// Mitsubishi GX Works2 project: GCP-75A2RB-(SECS)20220112   PLC: Q03UDV

PROGRAM 01INITI
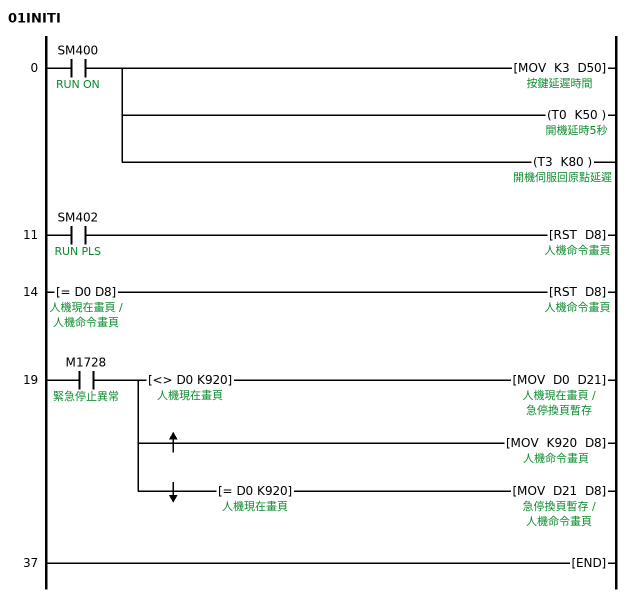
0     LD      SM400  ; RUN ON
      MOV     K3 D50  ; 按鍵延遲時間
      OUT     T0 K50  ; 開機延時5秒
      OUT     T3 K80  ; 開機伺服回原點延遲
11    LD      SM402  ; RUN PLS
      RST     D8  ; 人機命令畫頁
14    LD=     D0 D8  ; 人機現在畫頁 / 人機命令畫頁
      RST     D8  ; 人機命令畫頁
19    LD      M1728  ; 緊急停止異常
      MPS
      AND<>   D0 K920  ; 人機現在畫頁
      MOV     D0 D21  ; 急停換頁暫存
      MRD
      MEP
      MOV     K920 D8
      MPP
      MEF
      AND=    D0 K920  ; 人機現在畫頁
      MOV     D21 D8
37    END
END_PROGRAM

PROGRAM 02FUNC
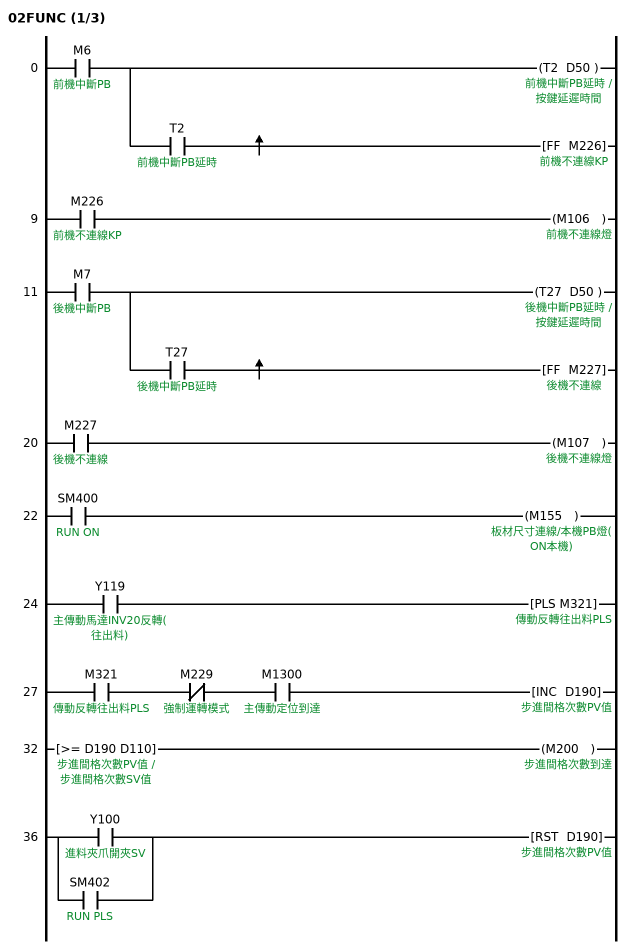
0     LD      M6  ; 前機中斷PB
      OUT     T2 D50  ; 前機中斷PB延時 / 按鍵延遲時間
      AND     T2  ; 前機中斷PB延時
      MEP
      FF      M226  ; 前機不連線KP
9     LD      M226  ; 前機不連線KP
      OUT     M106  ; 前機不連線燈
11    LD      M7  ; 後機中斷PB
      OUT     T27 D50  ; 後機中斷PB延時 / 按鍵延遲時間
      AND     T27  ; 後機中斷PB延時
      MEP
      FF      M227  ; 後機不連線
20    LD      M227  ; 後機不連線
      OUT     M107  ; 後機不連線燈
22    LD      SM400  ; RUN ON
      OUT     M155  ; 板材尺寸連線/本機PB燈(ON本機)
24    LD      Y119  ; 主傳動馬達INV20反轉(往出料)
      PLS     M321  ; 傳動反轉往出料PLS
27    LD      M321  ; 傳動反轉往出料PLS
      ANI     M229  ; 強制運轉模式
      AND     M1300  ; 主傳動定位到達
      INC     D190  ; 步進間格次數PV值
32    LD>=    D190 D110  ; 步進間格次數PV值 / 步進間格次數SV值
      OUT     M200  ; 步進間格次數到達
36    LD      Y100  ; 進料夾爪開夾SV
      OR      SM402  ; RUN PLS
      RST     D190  ; 步進間格次數PV值
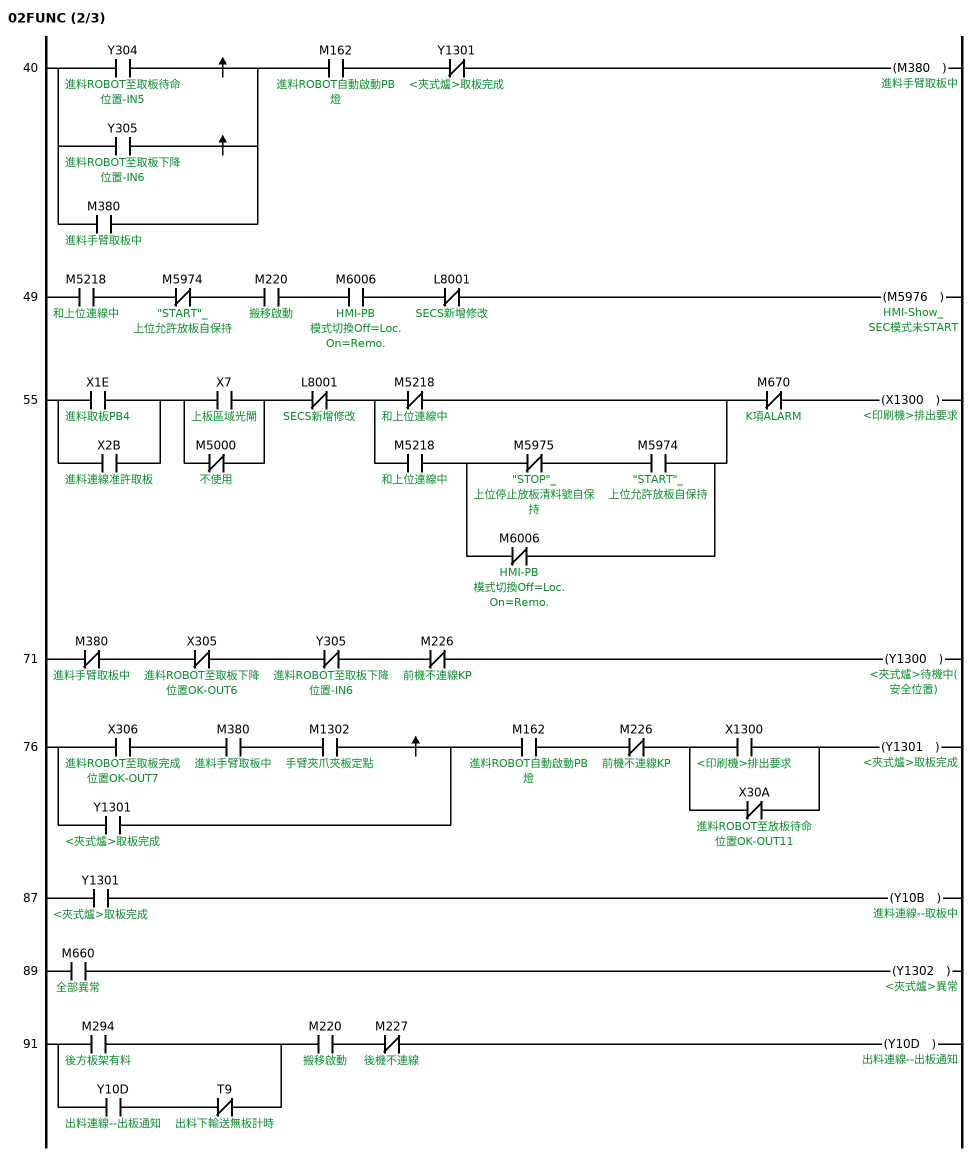
40    LD      Y304  ; 進料ROBOT至取板待命位置-IN5
      MEP
      LD      Y305  ; 進料ROBOT至取板下降位置-IN6
      MEP
      ORB
      OR      M380  ; 進料手臂取板中
      AND     M162  ; 進料ROBOT自動啟動PB燈
      ANI     Y1301  ; <夾式爐>取板完成
      OUT     M380  ; 進料手臂取板中
49    LD      M5218  ; 和上位連線中
      ANI     M5974  ; "START"_上位允許放板自保持
      AND     M220  ; 搬移啟動
      AND     M6006  ; HMI-PB  模式切換Off=Loc.On=Remo.
      ANI     L8001  ; SECS新增修改
      OUT     M5976  ; HMI-Show_SEC模式未START
55    LD      X1E  ; 進料取板PB4
      OR      X2B  ; 進料連線准許取板
      LD      X7  ; 上板區域光閘
      ORI     M5000  ; 不使用
      ANB
      ANI     L8001  ; SECS新增修改
      LDI     M5218  ; 和上位連線中
      LD      M5218  ; 和上位連線中
      LDI     M5975  ; "STOP"_ 上位停止放板清料號自保持
      AND     M5974  ; "START"_上位允許放板自保持
      ORI     M6006  ; HMI-PB  模式切換Off=Loc.On=Remo.
      ANB
      ORB
      ANB
      ANI     M670  ; K項ALARM
      OUT     X1300  ; <印刷機>排出要求
71    LDI     M380  ; 進料手臂取板中
      ANI     X305  ; 進料ROBOT至取板下降位置OK-OUT6
      ANI     Y305  ; 進料ROBOT至取板下降位置-IN6
      ANI     M226  ; 前機不連線KP
      OUT     Y1300  ; <夾式爐>待機中(安全位置)
76    LD      X306  ; 進料ROBOT至取板完成位置OK-OUT7
      AND     M380  ; 進料手臂取板中
      AND     M1302  ; 手臂夾爪夾板定點
      MEP
      OR      Y1301  ; <夾式爐>取板完成
      AND     M162  ; 進料ROBOT自動啟動PB燈
      ANI     M226  ; 前機不連線KP
      LD      X1300  ; <印刷機>排出要求
      ORI     X30A  ; 進料ROBOT至放板待命位置OK-OUT11
      ANB
      OUT     Y1301  ; <夾式爐>取板完成
87    LD      Y1301  ; <夾式爐>取板完成
      OUT     Y10B  ; 進料連線--取板中
89    LD      M660  ; 全部異常
      OUT     Y1302  ; <夾式爐>異常
91    LD      M294  ; 後方板架有料
      LD      Y10D  ; 出料連線--出板通知
      ANI     T9  ; 出料下輸送無板計時
      ORB
      AND     M220  ; 搬移啟動
      ANI     M227  ; 後機不連線
      OUT     Y10D  ; 出料連線--出板通知
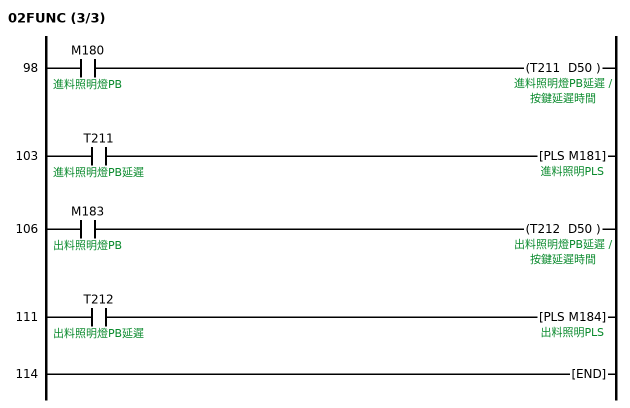
98    LD      M180  ; 進料照明燈PB
      OUT     T211 D50  ; 進料照明燈PB延遲 / 按鍵延遲時間
103   LD      T211  ; 進料照明燈PB延遲
      PLS     M181  ; 進料照明PLS
106   LD      M183  ; 出料照明燈PB
      OUT     T212 D50  ; 出料照明燈PB延遲 / 按鍵延遲時間
111   LD      T212  ; 出料照明燈PB延遲
      PLS     M184  ; 出料照明PLS
114   END
END_PROGRAM

PROGRAM 03ORIGIN
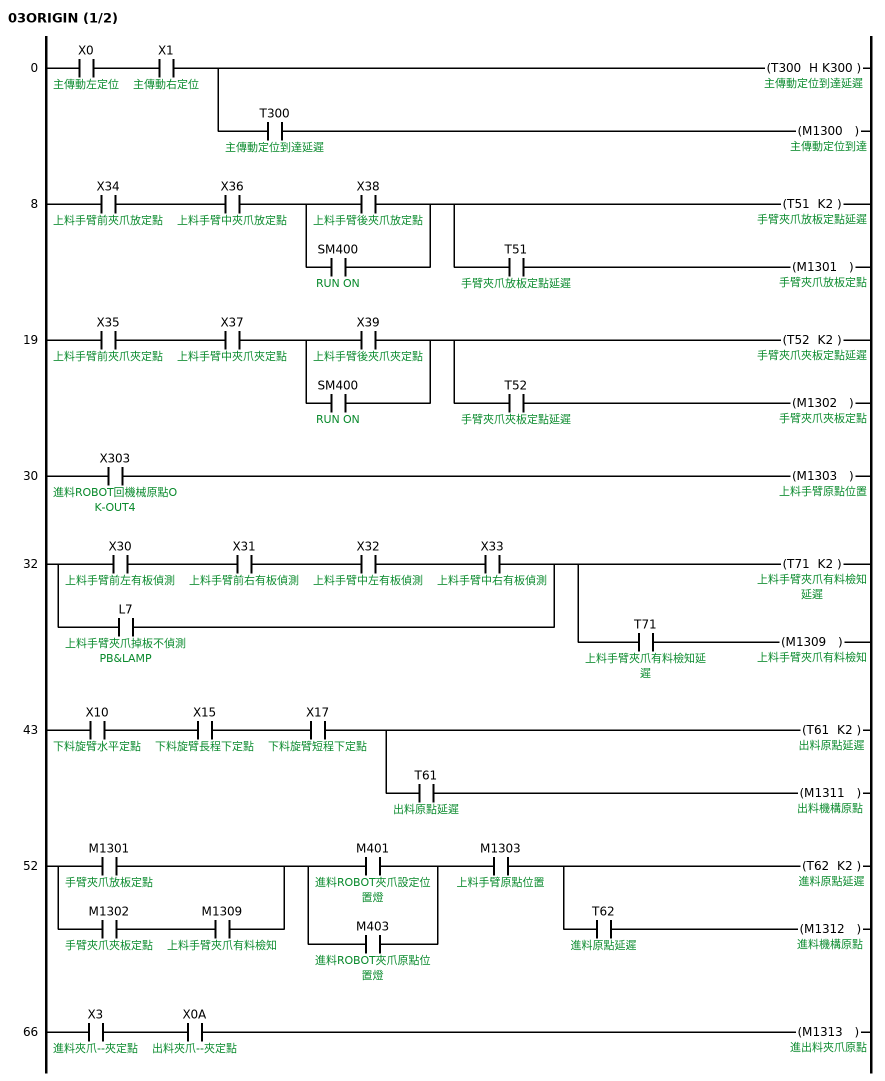
0     LD      X0  ; 主傳動左定位
      AND     X1  ; 主傳動右定位
      OUTH    T300 K300  ; 主傳動定位到達延遲
      AND     T300  ; 主傳動定位到達延遲
      OUT     M1300  ; 主傳動定位到達
8     LD      X34  ; 上料手臂前夾爪放定點
      AND     X36  ; 上料手臂中夾爪放定點
      LD      X38  ; 上料手臂後夾爪放定點
      OR      SM400  ; RUN ON
      ANB
      OUT     T51 K2  ; 手臂夾爪放板定點延遲
      AND     T51  ; 手臂夾爪放板定點延遲
      OUT     M1301  ; 手臂夾爪放板定點
19    LD      X35  ; 上料手臂前夾爪夾定點
      AND     X37  ; 上料手臂中夾爪夾定點
      LD      X39  ; 上料手臂後夾爪夾定點
      OR      SM400  ; RUN ON
      ANB
      OUT     T52 K2  ; 手臂夾爪夾板定點延遲
      AND     T52  ; 手臂夾爪夾板定點延遲
      OUT     M1302  ; 手臂夾爪夾板定點
30    LD      X303  ; 進料ROBOT回機械原點OK-OUT4
      OUT     M1303  ; 上料手臂原點位置
32    LD      X30  ; 上料手臂前左有板偵測
      AND     X31  ; 上料手臂前右有板偵測
      AND     X32  ; 上料手臂中左有板偵測
      AND     X33  ; 上料手臂中右有板偵測
      OR      L7  ; 上料手臂夾爪掉板不偵測PB&LAMP
      OUT     T71 K2  ; 上料手臂夾爪有料檢知延遲
      AND     T71  ; 上料手臂夾爪有料檢知延遲
      OUT     M1309  ; 上料手臂夾爪有料檢知
43    LD      X10  ; 下料旋臂水平定點
      AND     X15  ; 下料旋臂長程下定點
      AND     X17  ; 下料旋臂短程下定點
      OUT     T61 K2  ; 出料原點延遲
      AND     T61  ; 出料原點延遲
      OUT     M1311  ; 出料機構原點
52    LD      M1301  ; 手臂夾爪放板定點
      LD      M1302  ; 手臂夾爪夾板定點
      AND     M1309  ; 上料手臂夾爪有料檢知
      ORB
      LD      M401  ; 進料ROBOT夾爪設定位置燈
      OR      M403  ; 進料ROBOT夾爪原點位置燈
      ANB
      AND     M1303  ; 上料手臂原點位置
      OUT     T62 K2  ; 進料原點延遲
      AND     T62  ; 進料原點延遲
      OUT     M1312  ; 進料機構原點
66    LD      X3  ; 進料夾爪--夾定點
      AND     X0A  ; 出料夾爪--夾定點
      OUT     M1313  ; 進出料夾爪原點
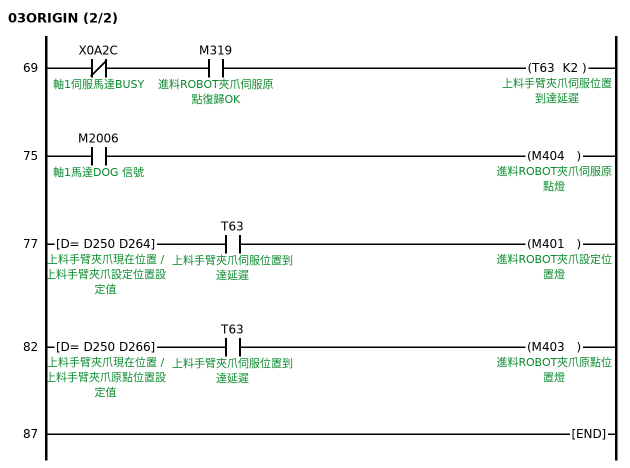
69    LDI     X0A2C  ; 軸1伺服馬達BUSY
      AND     M319  ; 進料ROBOT夾爪伺服原點復歸OK
      OUT     T63 K2  ; 上料手臂夾爪伺服位置到達延遲
75    LD      M2006  ; 軸1馬達DOG 信號
      OUT     M404  ; 進料ROBOT夾爪伺服原點燈
77    LDD=    D250 D264  ; 上料手臂夾爪現在位置 / 上料手臂夾爪設定位置設定值
      AND     T63  ; 上料手臂夾爪伺服位置到達延遲
      OUT     M401  ; 進料ROBOT夾爪設定位置燈
82    LDD=    D250 D266  ; 上料手臂夾爪現在位置 / 上料手臂夾爪原點位置設定值
      AND     T63  ; 上料手臂夾爪伺服位置到達延遲
      OUT     M403  ; 進料ROBOT夾爪原點位置燈
87    END
END_PROGRAM

PROGRAM 04LOAD
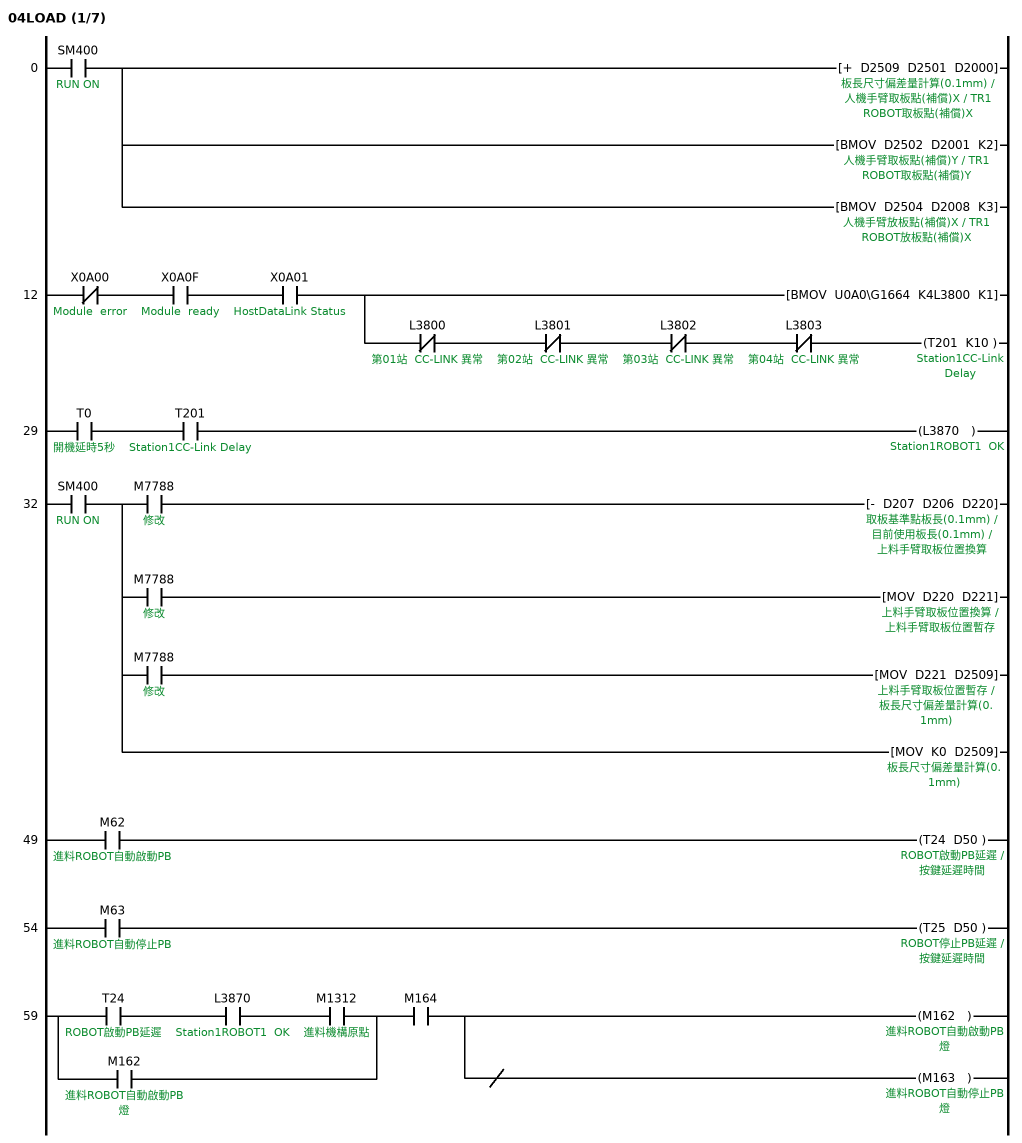
0     LD      SM400  ; RUN ON
      +       D2509 D2501 D2000  ; 板長尺寸偏差量計算(0.1mm) / 人機手臂取板點(補償)X / TR1 ROBOT取板點(補償)X
      BMOV    D2502 D2001 K2  ; 人機手臂取板點(補償)Y / TR1 ROBOT取板點(補償)Y
      BMOV    D2504 D2008 K3  ; 人機手臂放板點(補償)X / TR1 ROBOT放板點(補償)X
12    LDI     X0A00  ; Module  error
      AND     X0A0F  ; Module  ready
      AND     X0A01  ; HostDataLink Status
      BMOV    U0A0\G1664 K4L3800 K1  ; 第01站  CC-LINK 異常
      ANI     L3800  ; 第01站  CC-LINK 異常
      ANI     L3801  ; 第02站  CC-LINK 異常
      ANI     L3802  ; 第03站  CC-LINK 異常
      ANI     L3803  ; 第04站  CC-LINK 異常
      OUT     T201 K10  ; Station1CC-Link Delay
29    LD      T0  ; 開機延時5秒
      AND     T201  ; Station1CC-Link Delay
      OUT     L3870  ; Station1ROBOT1  OK
32    LD      SM400  ; RUN ON
      MPS
      AND     M7788  ; 修改
      -       D207 D206 D220  ; 取板基準點板長(0.1mm) / 目前使用板長(0.1mm) / 上料手臂取板位置換算
      MRD
      AND     M7788  ; 修改
      MOV     D220 D221  ; 上料手臂取板位置暫存
      MRD
      AND     M7788  ; 修改
      MOV     D221 D2509
      MPP
      MOV     K0 D2509
49    LD      M62  ; 進料ROBOT自動啟動PB
      OUT     T24 D50  ; ROBOT啟動PB延遲 / 按鍵延遲時間
54    LD      M63  ; 進料ROBOT自動停止PB
      OUT     T25 D50  ; ROBOT停止PB延遲 / 按鍵延遲時間
59    LD      T24  ; ROBOT啟動PB延遲
      AND     L3870  ; Station1ROBOT1  OK
      AND     M1312  ; 進料機構原點
      OR      M162  ; 進料ROBOT自動啟動PB燈
      AND     M164
      OUT     M162  ; 進料ROBOT自動啟動PB燈
      INV
      OUT     M163  ; 進料ROBOT自動停止PB燈
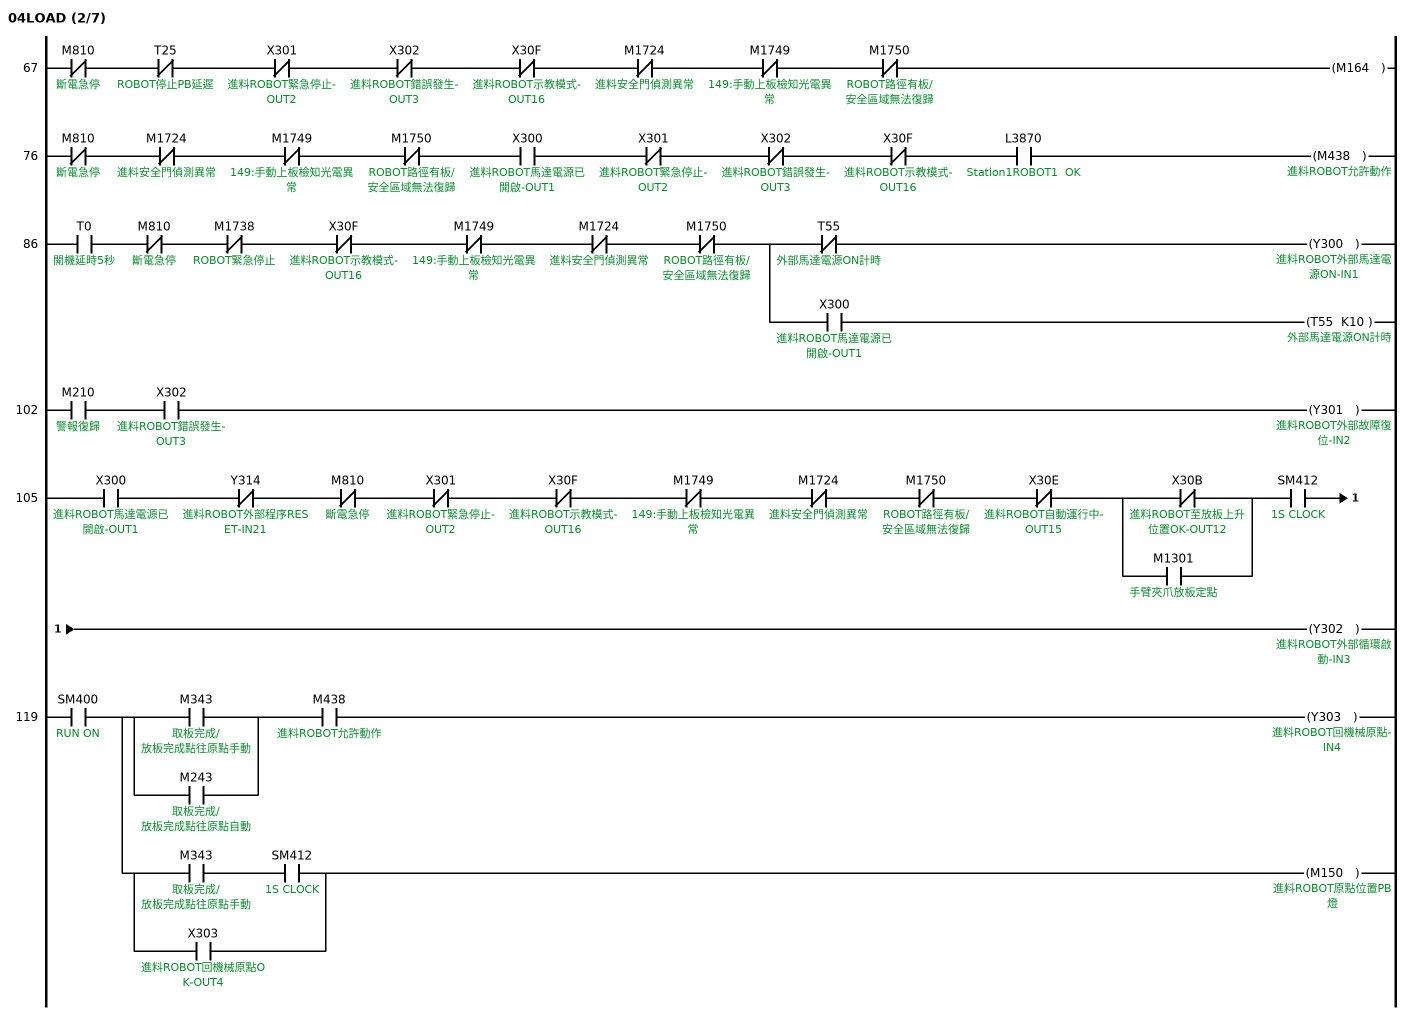
67    LDI     M810  ; 斷電急停
      ANI     T25  ; ROBOT停止PB延遲
      ANI     X301  ; 進料ROBOT緊急停止-OUT2
      ANI     X302  ; 進料ROBOT錯誤發生-OUT3
      ANI     X30F  ; 進料ROBOT示教模式-OUT16
      ANI     M1724  ; 進料安全門偵測異常
      ANI     M1749  ; 149:手動上板檢知光電異常
      ANI     M1750  ; ROBOT路徑有板/安全區域無法復歸
      OUT     M164
76    LDI     M810  ; 斷電急停
      ANI     M1724  ; 進料安全門偵測異常
      ANI     M1749  ; 149:手動上板檢知光電異常
      ANI     M1750  ; ROBOT路徑有板/安全區域無法復歸
      AND     X300  ; 進料ROBOT馬達電源已開啟-OUT1
      ANI     X301  ; 進料ROBOT緊急停止-OUT2
      ANI     X302  ; 進料ROBOT錯誤發生-OUT3
      ANI     X30F  ; 進料ROBOT示教模式-OUT16
      AND     L3870  ; Station1ROBOT1  OK
      OUT     M438  ; 進料ROBOT允許動作
86    LD      T0  ; 開機延時5秒
      ANI     M810  ; 斷電急停
      ANI     M1738  ; ROBOT緊急停止
      ANI     X30F  ; 進料ROBOT示教模式-OUT16
      ANI     M1749  ; 149:手動上板檢知光電異常
      ANI     M1724  ; 進料安全門偵測異常
      ANI     M1750  ; ROBOT路徑有板/安全區域無法復歸
      MPS
      ANI     T55  ; 外部馬達電源ON計時
      OUT     Y300  ; 進料ROBOT外部馬達電源ON-IN1
      MPP
      AND     X300  ; 進料ROBOT馬達電源已開啟-OUT1
      OUT     T55 K10  ; 外部馬達電源ON計時
102   LD      M210  ; 警報復歸
      AND     X302  ; 進料ROBOT錯誤發生-OUT3
      OUT     Y301  ; 進料ROBOT外部故障復位-IN2
105   LD      X300  ; 進料ROBOT馬達電源已開啟-OUT1
      ANI     Y314  ; 進料ROBOT外部程序RESET-IN21
      ANI     M810  ; 斷電急停
      ANI     X301  ; 進料ROBOT緊急停止-OUT2
      ANI     X30F  ; 進料ROBOT示教模式-OUT16
      ANI     M1749  ; 149:手動上板檢知光電異常
      ANI     M1724  ; 進料安全門偵測異常
      ANI     M1750  ; ROBOT路徑有板/安全區域無法復歸
      ANI     X30E  ; 進料ROBOT自動運行中-OUT15
      LDI     X30B  ; 進料ROBOT至放板上升位置OK-OUT12
      OR      M1301  ; 手臂夾爪放板定點
      ANB
      AND     SM412  ; 1S CLOCK
      OUT     Y302  ; 進料ROBOT外部循環啟動-IN3
119   LD      SM400  ; RUN ON
      MPS
      LD      M343  ; 取板完成/放板完成點往原點手動
      OR      M243  ; 取板完成/放板完成點往原點自動
      ANB
      AND     M438  ; 進料ROBOT允許動作
      OUT     Y303  ; 進料ROBOT回機械原點-IN4
      MPP
      LD      M343  ; 取板完成/放板完成點往原點手動
      AND     SM412  ; 1S CLOCK
      OR      X303  ; 進料ROBOT回機械原點OK-OUT4
      ANB
      OUT     M150  ; 進料ROBOT原點位置PB燈
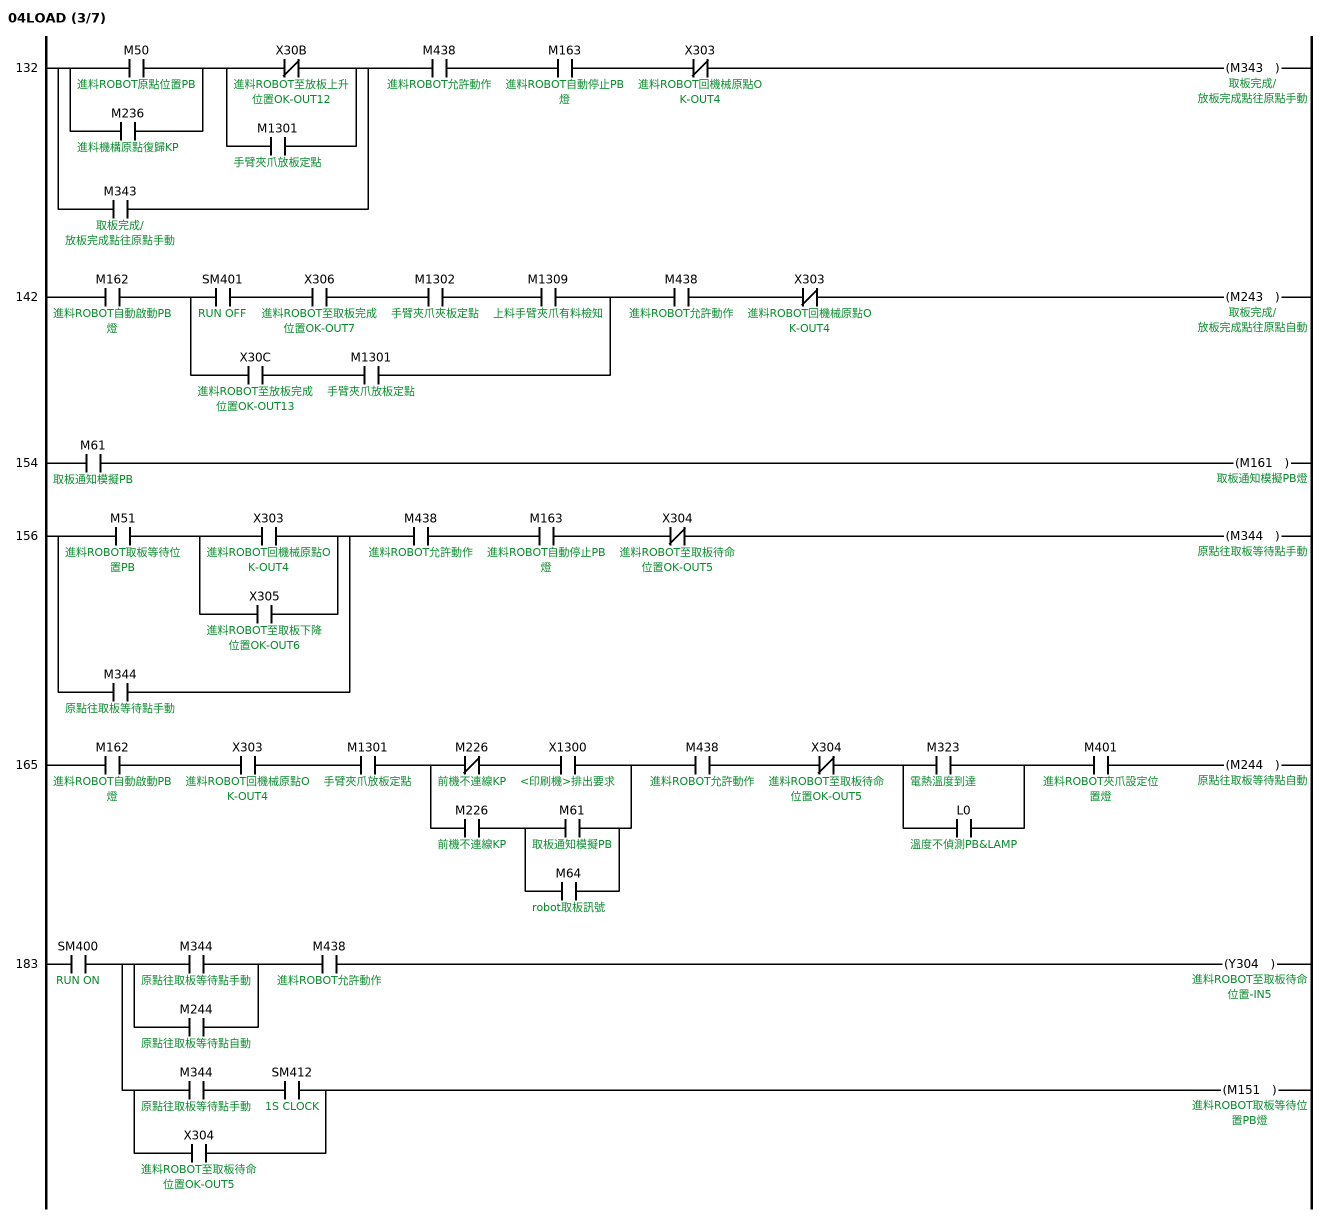
132   LD      M50  ; 進料ROBOT原點位置PB
      OR      M236  ; 進料機構原點復歸KP
      LDI     X30B  ; 進料ROBOT至放板上升位置OK-OUT12
      OR      M1301  ; 手臂夾爪放板定點
      ANB
      OR      M343  ; 取板完成/放板完成點往原點手動
      AND     M438  ; 進料ROBOT允許動作
      AND     M163  ; 進料ROBOT自動停止PB燈
      ANI     X303  ; 進料ROBOT回機械原點OK-OUT4
      OUT     M343  ; 取板完成/放板完成點往原點手動
142   LD      M162  ; 進料ROBOT自動啟動PB燈
      LD      SM401  ; RUN OFF
      AND     X306  ; 進料ROBOT至取板完成位置OK-OUT7
      AND     M1302  ; 手臂夾爪夾板定點
      AND     M1309  ; 上料手臂夾爪有料檢知
      LD      X30C  ; 進料ROBOT至放板完成位置OK-OUT13
      AND     M1301  ; 手臂夾爪放板定點
      ORB
      ANB
      AND     M438  ; 進料ROBOT允許動作
      ANI     X303  ; 進料ROBOT回機械原點OK-OUT4
      OUT     M243  ; 取板完成/放板完成點往原點自動
154   LD      M61  ; 取板通知模擬PB
      OUT     M161  ; 取板通知模擬PB燈
156   LD      M51  ; 進料ROBOT取板等待位置PB
      LD      X303  ; 進料ROBOT回機械原點OK-OUT4
      OR      X305  ; 進料ROBOT至取板下降位置OK-OUT6
      ANB
      OR      M344  ; 原點往取板等待點手動
      AND     M438  ; 進料ROBOT允許動作
      AND     M163  ; 進料ROBOT自動停止PB燈
      ANI     X304  ; 進料ROBOT至取板待命位置OK-OUT5
      OUT     M344  ; 原點往取板等待點手動
165   LD      M162  ; 進料ROBOT自動啟動PB燈
      AND     X303  ; 進料ROBOT回機械原點OK-OUT4
      AND     M1301  ; 手臂夾爪放板定點
      LDI     M226  ; 前機不連線KP
      AND     X1300  ; <印刷機>排出要求
      LD      M226  ; 前機不連線KP
      LD      M61  ; 取板通知模擬PB
      OR      M64  ; robot取板訊號
      ANB
      ORB
      ANB
      AND     M438  ; 進料ROBOT允許動作
      ANI     X304  ; 進料ROBOT至取板待命位置OK-OUT5
      LD      M323  ; 電熱溫度到達
      OR      L0  ; 溫度不偵測PB&LAMP
      ANB
      AND     M401  ; 進料ROBOT夾爪設定位置燈
      OUT     M244  ; 原點往取板等待點自動
183   LD      SM400  ; RUN ON
      MPS
      LD      M344  ; 原點往取板等待點手動
      OR      M244  ; 原點往取板等待點自動
      ANB
      AND     M438  ; 進料ROBOT允許動作
      OUT     Y304  ; 進料ROBOT至取板待命位置-IN5
      MPP
      LD      M344  ; 原點往取板等待點手動
      AND     SM412  ; 1S CLOCK
      OR      X304  ; 進料ROBOT至取板待命位置OK-OUT5
      ANB
      OUT     M151  ; 進料ROBOT取板等待位置PB燈
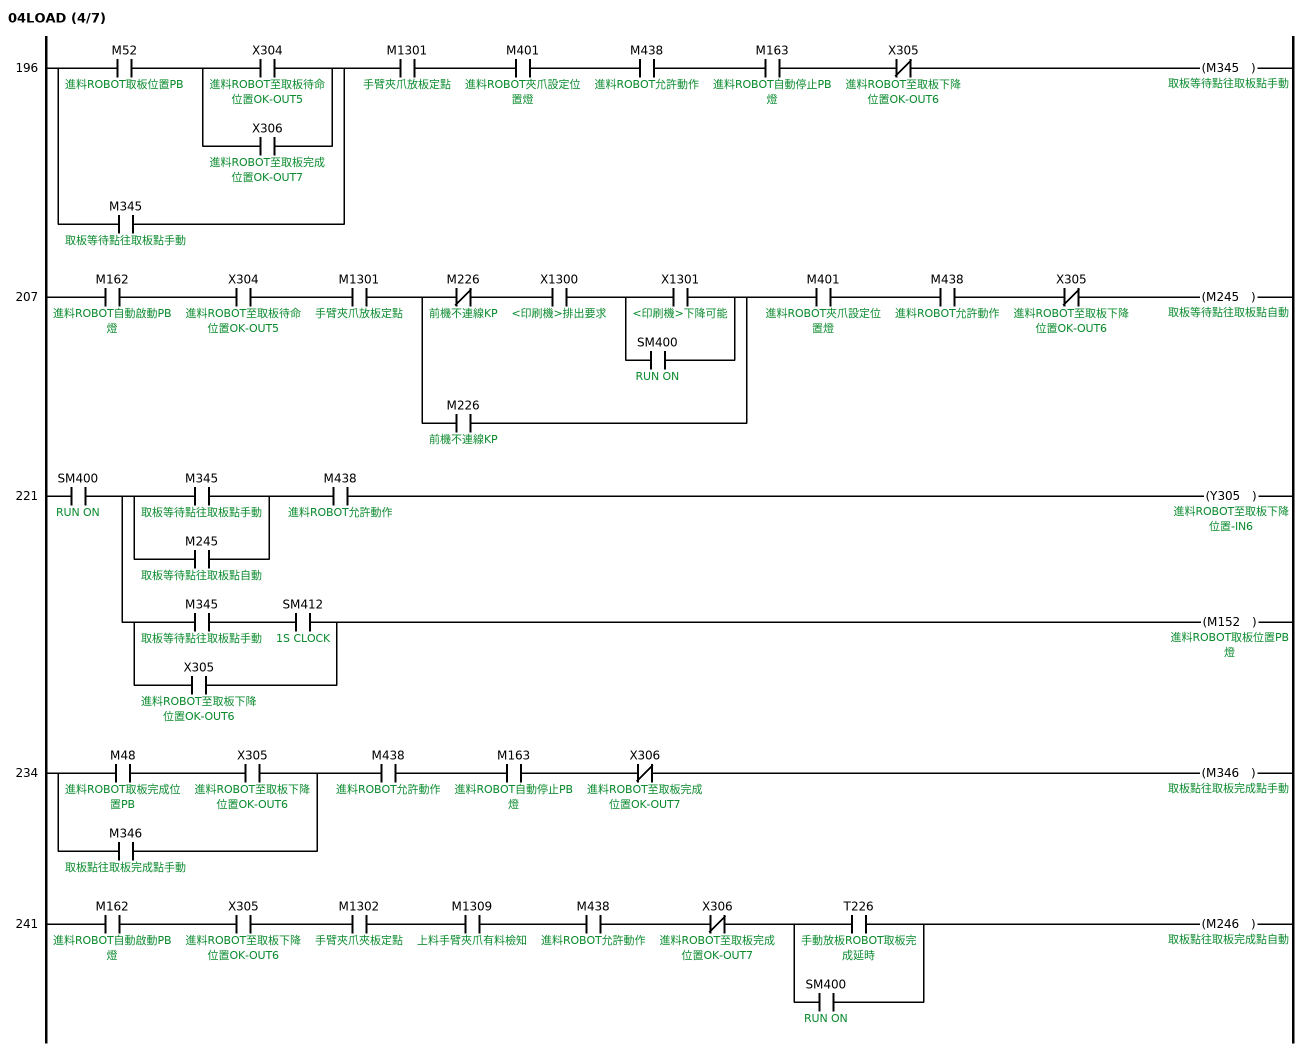
196   LD      M52  ; 進料ROBOT取板位置PB
      LD      X304  ; 進料ROBOT至取板待命位置OK-OUT5
      OR      X306  ; 進料ROBOT至取板完成位置OK-OUT7
      ANB
      OR      M345  ; 取板等待點往取板點手動
      AND     M1301  ; 手臂夾爪放板定點
      AND     M401  ; 進料ROBOT夾爪設定位置燈
      AND     M438  ; 進料ROBOT允許動作
      AND     M163  ; 進料ROBOT自動停止PB燈
      ANI     X305  ; 進料ROBOT至取板下降位置OK-OUT6
      OUT     M345  ; 取板等待點往取板點手動
207   LD      M162  ; 進料ROBOT自動啟動PB燈
      AND     X304  ; 進料ROBOT至取板待命位置OK-OUT5
      AND     M1301  ; 手臂夾爪放板定點
      LDI     M226  ; 前機不連線KP
      AND     X1300  ; <印刷機>排出要求
      LD      X1301  ; <印刷機>下降可能
      OR      SM400  ; RUN ON
      ANB
      OR      M226  ; 前機不連線KP
      ANB
      AND     M401  ; 進料ROBOT夾爪設定位置燈
      AND     M438  ; 進料ROBOT允許動作
      ANI     X305  ; 進料ROBOT至取板下降位置OK-OUT6
      OUT     M245  ; 取板等待點往取板點自動
221   LD      SM400  ; RUN ON
      MPS
      LD      M345  ; 取板等待點往取板點手動
      OR      M245  ; 取板等待點往取板點自動
      ANB
      AND     M438  ; 進料ROBOT允許動作
      OUT     Y305  ; 進料ROBOT至取板下降位置-IN6
      MPP
      LD      M345  ; 取板等待點往取板點手動
      AND     SM412  ; 1S CLOCK
      OR      X305  ; 進料ROBOT至取板下降位置OK-OUT6
      ANB
      OUT     M152  ; 進料ROBOT取板位置PB燈
234   LD      M48  ; 進料ROBOT取板完成位置PB
      AND     X305  ; 進料ROBOT至取板下降位置OK-OUT6
      OR      M346  ; 取板點往取板完成點手動
      AND     M438  ; 進料ROBOT允許動作
      AND     M163  ; 進料ROBOT自動停止PB燈
      ANI     X306  ; 進料ROBOT至取板完成位置OK-OUT7
      OUT     M346  ; 取板點往取板完成點手動
241   LD      M162  ; 進料ROBOT自動啟動PB燈
      AND     X305  ; 進料ROBOT至取板下降位置OK-OUT6
      AND     M1302  ; 手臂夾爪夾板定點
      AND     M1309  ; 上料手臂夾爪有料檢知
      AND     M438  ; 進料ROBOT允許動作
      ANI     X306  ; 進料ROBOT至取板完成位置OK-OUT7
      LD      T226  ; 手動放板ROBOT取板完成延時
      OR      SM400  ; RUN ON
      ANB
      OUT     M246  ; 取板點往取板完成點自動
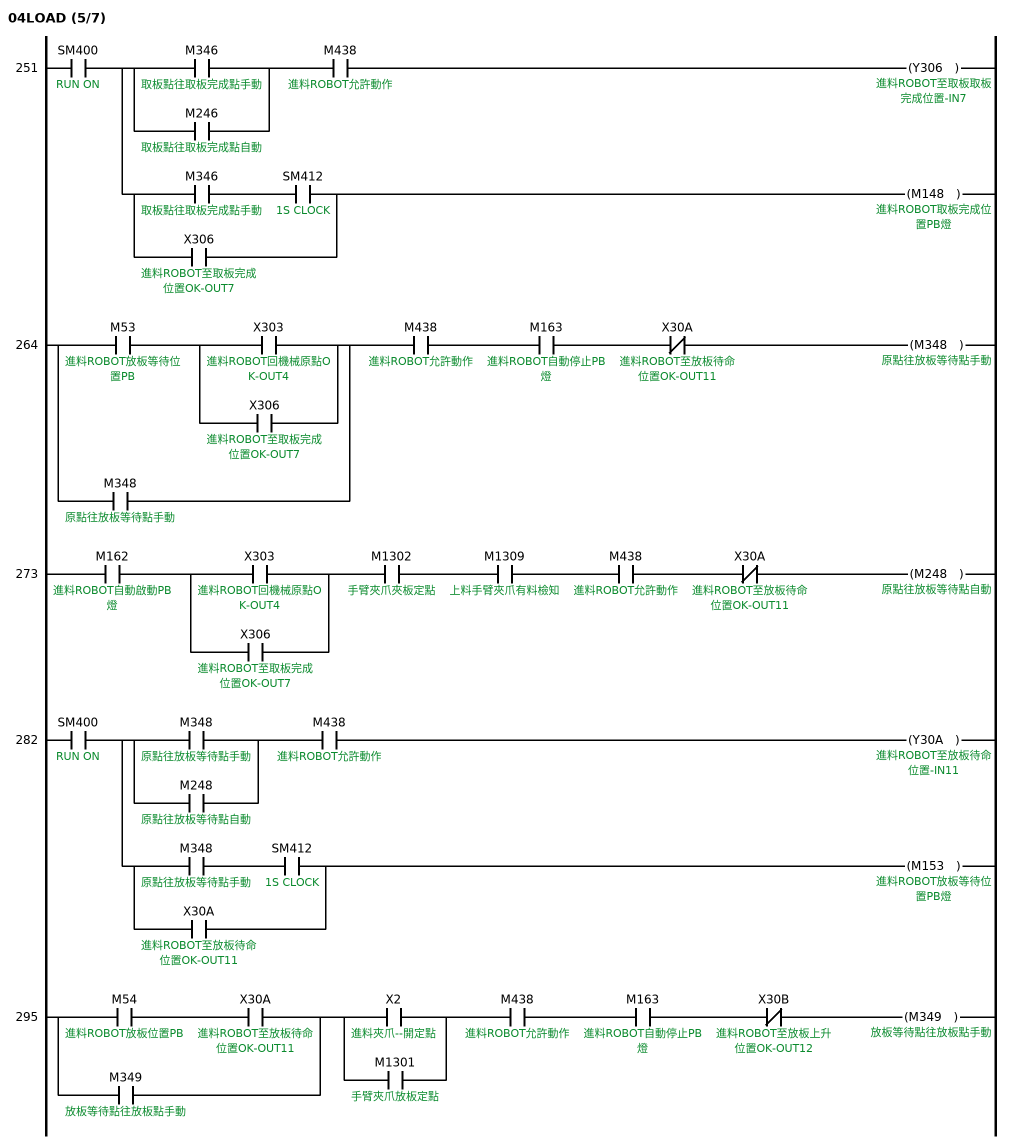
251   LD      SM400  ; RUN ON
      MPS
      LD      M346  ; 取板點往取板完成點手動
      OR      M246  ; 取板點往取板完成點自動
      ANB
      AND     M438  ; 進料ROBOT允許動作
      OUT     Y306  ; 進料ROBOT至取板取板完成位置-IN7
      MPP
      LD      M346  ; 取板點往取板完成點手動
      AND     SM412  ; 1S CLOCK
      OR      X306  ; 進料ROBOT至取板完成位置OK-OUT7
      ANB
      OUT     M148  ; 進料ROBOT取板完成位置PB燈
264   LD      M53  ; 進料ROBOT放板等待位置PB
      LD      X303  ; 進料ROBOT回機械原點OK-OUT4
      OR      X306  ; 進料ROBOT至取板完成位置OK-OUT7
      ANB
      OR      M348  ; 原點往放板等待點手動
      AND     M438  ; 進料ROBOT允許動作
      AND     M163  ; 進料ROBOT自動停止PB燈
      ANI     X30A  ; 進料ROBOT至放板待命位置OK-OUT11
      OUT     M348  ; 原點往放板等待點手動
273   LD      M162  ; 進料ROBOT自動啟動PB燈
      LD      X303  ; 進料ROBOT回機械原點OK-OUT4
      OR      X306  ; 進料ROBOT至取板完成位置OK-OUT7
      ANB
      AND     M1302  ; 手臂夾爪夾板定點
      AND     M1309  ; 上料手臂夾爪有料檢知
      AND     M438  ; 進料ROBOT允許動作
      ANI     X30A  ; 進料ROBOT至放板待命位置OK-OUT11
      OUT     M248  ; 原點往放板等待點自動
282   LD      SM400  ; RUN ON
      MPS
      LD      M348  ; 原點往放板等待點手動
      OR      M248  ; 原點往放板等待點自動
      ANB
      AND     M438  ; 進料ROBOT允許動作
      OUT     Y30A  ; 進料ROBOT至放板待命位置-IN11
      MPP
      LD      M348  ; 原點往放板等待點手動
      AND     SM412  ; 1S CLOCK
      OR      X30A  ; 進料ROBOT至放板待命位置OK-OUT11
      ANB
      OUT     M153  ; 進料ROBOT放板等待位置PB燈
295   LD      M54  ; 進料ROBOT放板位置PB
      AND     X30A  ; 進料ROBOT至放板待命位置OK-OUT11
      OR      M349  ; 放板等待點往放板點手動
      LD      X2  ; 進料夾爪--開定點
      OR      M1301  ; 手臂夾爪放板定點
      ANB
      AND     M438  ; 進料ROBOT允許動作
      AND     M163  ; 進料ROBOT自動停止PB燈
      ANI     X30B  ; 進料ROBOT至放板上升位置OK-OUT12
      OUT     M349  ; 放板等待點往放板點手動
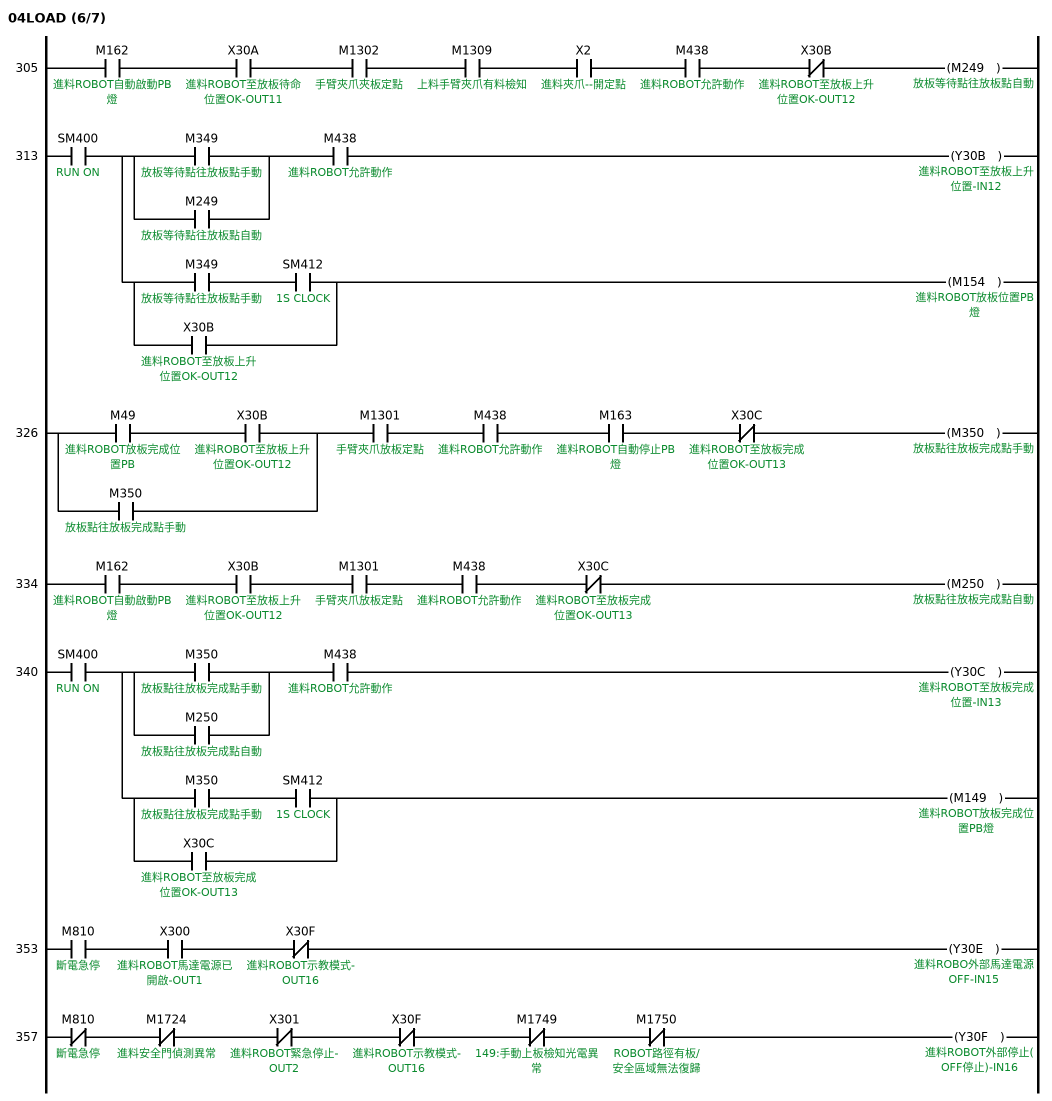
305   LD      M162  ; 進料ROBOT自動啟動PB燈
      AND     X30A  ; 進料ROBOT至放板待命位置OK-OUT11
      AND     M1302  ; 手臂夾爪夾板定點
      AND     M1309  ; 上料手臂夾爪有料檢知
      AND     X2  ; 進料夾爪--開定點
      AND     M438  ; 進料ROBOT允許動作
      ANI     X30B  ; 進料ROBOT至放板上升位置OK-OUT12
      OUT     M249  ; 放板等待點往放板點自動
313   LD      SM400  ; RUN ON
      MPS
      LD      M349  ; 放板等待點往放板點手動
      OR      M249  ; 放板等待點往放板點自動
      ANB
      AND     M438  ; 進料ROBOT允許動作
      OUT     Y30B  ; 進料ROBOT至放板上升位置-IN12
      MPP
      LD      M349  ; 放板等待點往放板點手動
      AND     SM412  ; 1S CLOCK
      OR      X30B  ; 進料ROBOT至放板上升位置OK-OUT12
      ANB
      OUT     M154  ; 進料ROBOT放板位置PB燈
326   LD      M49  ; 進料ROBOT放板完成位置PB
      AND     X30B  ; 進料ROBOT至放板上升位置OK-OUT12
      OR      M350  ; 放板點往放板完成點手動
      AND     M1301  ; 手臂夾爪放板定點
      AND     M438  ; 進料ROBOT允許動作
      AND     M163  ; 進料ROBOT自動停止PB燈
      ANI     X30C  ; 進料ROBOT至放板完成位置OK-OUT13
      OUT     M350  ; 放板點往放板完成點手動
334   LD      M162  ; 進料ROBOT自動啟動PB燈
      AND     X30B  ; 進料ROBOT至放板上升位置OK-OUT12
      AND     M1301  ; 手臂夾爪放板定點
      AND     M438  ; 進料ROBOT允許動作
      ANI     X30C  ; 進料ROBOT至放板完成位置OK-OUT13
      OUT     M250  ; 放板點往放板完成點自動
340   LD      SM400  ; RUN ON
      MPS
      LD      M350  ; 放板點往放板完成點手動
      OR      M250  ; 放板點往放板完成點自動
      ANB
      AND     M438  ; 進料ROBOT允許動作
      OUT     Y30C  ; 進料ROBOT至放板完成位置-IN13
      MPP
      LD      M350  ; 放板點往放板完成點手動
      AND     SM412  ; 1S CLOCK
      OR      X30C  ; 進料ROBOT至放板完成位置OK-OUT13
      ANB
      OUT     M149  ; 進料ROBOT放板完成位置PB燈
353   LD      M810  ; 斷電急停
      AND     X300  ; 進料ROBOT馬達電源已開啟-OUT1
      ANI     X30F  ; 進料ROBOT示教模式-OUT16
      OUT     Y30E  ; 進料ROBO外部馬達電源OFF-IN15
357   LDI     M810  ; 斷電急停
      ANI     M1724  ; 進料安全門偵測異常
      ANI     X301  ; 進料ROBOT緊急停止-OUT2
      ANI     X30F  ; 進料ROBOT示教模式-OUT16
      ANI     M1749  ; 149:手動上板檢知光電異常
      ANI     M1750  ; ROBOT路徑有板/安全區域無法復歸
      OUT     Y30F  ; 進料ROBOT外部停止(OFF停止)-IN16
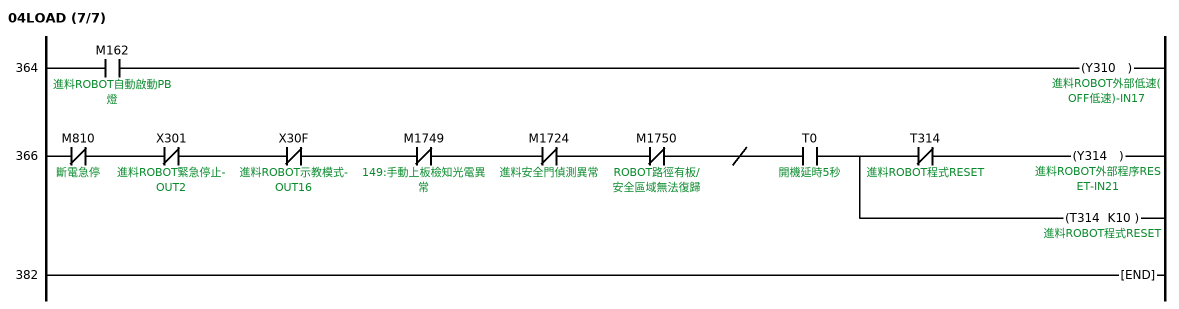
364   LD      M162  ; 進料ROBOT自動啟動PB燈
      OUT     Y310  ; 進料ROBOT外部低速(OFF低速)-IN17
366   LDI     M810  ; 斷電急停
      ANI     X301  ; 進料ROBOT緊急停止-OUT2
      ANI     X30F  ; 進料ROBOT示教模式-OUT16
      ANI     M1749  ; 149:手動上板檢知光電異常
      ANI     M1724  ; 進料安全門偵測異常
      ANI     M1750  ; ROBOT路徑有板/安全區域無法復歸
      INV
      AND     T0  ; 開機延時5秒
      MPS
      ANI     T314  ; 進料ROBOT程式RESET
      OUT     Y314  ; 進料ROBOT外部程序RESET-IN21
      MPP
      OUT     T314 K10  ; 進料ROBOT程式RESET
382   END
END_PROGRAM

PROGRAM 05LOADUP
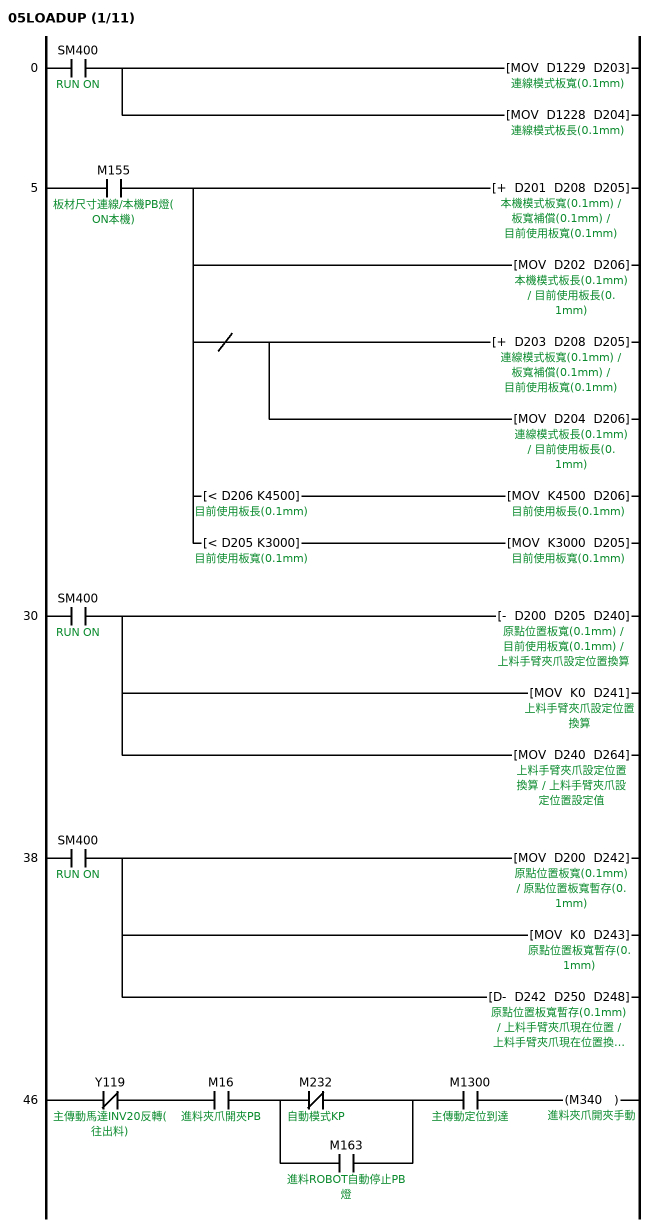
0     LD      SM400  ; RUN ON
      MOV     D1229 D203  ; 連線模式板寬(0.1mm)
      MOV     D1228 D204  ; 連線模式板長(0.1mm)
5     LD      M155  ; 板材尺寸連線/本機PB燈(ON本機)
      +       D201 D208 D205  ; 本機模式板寬(0.1mm) / 板寬補償(0.1mm) / 目前使用板寬(0.1mm)
      MOV     D202 D206  ; 本機模式板長(0.1mm) / 目前使用板長(0.1mm)
      MPS
      INV
      +       D203 D208 D205
      MOV     D204 D206
      MRD
      AND<    D206 K4500  ; 目前使用板長(0.1mm)
      MOV     K4500 D206
      MPP
      AND<    D205 K3000  ; 目前使用板寬(0.1mm)
      MOV     K3000 D205
30    LD      SM400  ; RUN ON
      -       D200 D205 D240  ; 原點位置板寬(0.1mm) / 上料手臂夾爪設定位置換算
      MOV     K0 D241  ; 上料手臂夾爪設定位置換算
      MOV     D240 D264  ; 上料手臂夾爪設定位置設定值
38    LD      SM400  ; RUN ON
      MOV     D200 D242  ; 原點位置板寬暫存(0.1mm)
      MOV     K0 D243  ; 原點位置板寬暫存(0.1mm)
      D-      D242 D250 D248  ; 上料手臂夾爪現在位置 / 上料手臂夾爪現在位置換算板寬
46    LDI     Y119  ; 主傳動馬達INV20反轉(往出料)
      AND     M16  ; 進料夾爪開夾PB
      LDI     M232  ; 自動模式KP
      OR      M163  ; 進料ROBOT自動停止PB燈
      ANB
      AND     M1300  ; 主傳動定位到達
      OUT     M340  ; 進料夾爪開夾手動
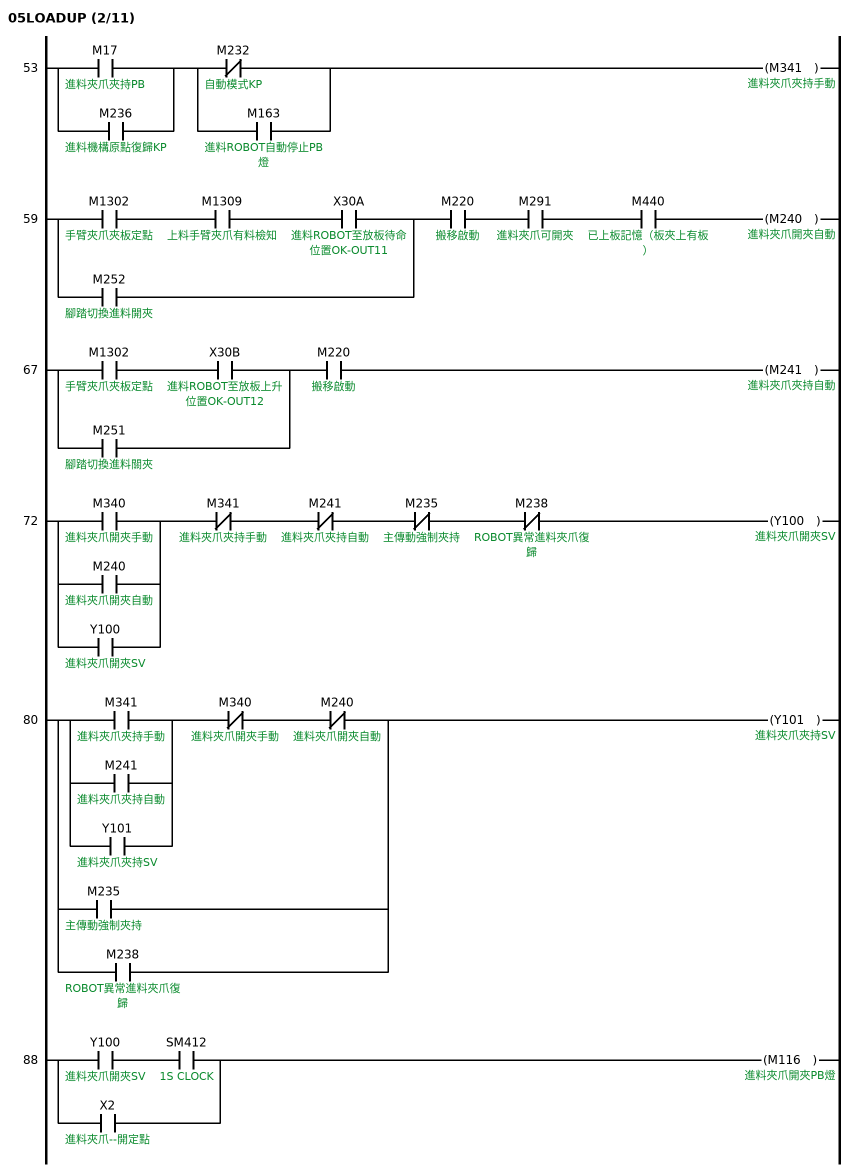
53    LD      M17  ; 進料夾爪夾持PB
      OR      M236  ; 進料機構原點復歸KP
      LDI     M232  ; 自動模式KP
      OR      M163  ; 進料ROBOT自動停止PB燈
      ANB
      OUT     M341  ; 進料夾爪夾持手動
59    LD      M1302  ; 手臂夾爪夾板定點
      AND     M1309  ; 上料手臂夾爪有料檢知
      AND     X30A  ; 進料ROBOT至放板待命位置OK-OUT11
      OR      M252  ; 腳踏切換進料開夾
      AND     M220  ; 搬移啟動
      AND     M291  ; 進料夾爪可開夾
      AND     M440  ; 已上板記憶（板夾上有板）
      OUT     M240  ; 進料夾爪開夾自動
67    LD      M1302  ; 手臂夾爪夾板定點
      AND     X30B  ; 進料ROBOT至放板上升位置OK-OUT12
      OR      M251  ; 腳踏切換進料關夾
      AND     M220  ; 搬移啟動
      OUT     M241  ; 進料夾爪夾持自動
72    LD      M340  ; 進料夾爪開夾手動
      OR      M240  ; 進料夾爪開夾自動
      OR      Y100  ; 進料夾爪開夾SV
      ANI     M341  ; 進料夾爪夾持手動
      ANI     M241  ; 進料夾爪夾持自動
      ANI     M235  ; 主傳動強制夾持
      ANI     M238  ; ROBOT異常進料夾爪復歸
      OUT     Y100  ; 進料夾爪開夾SV
80    LD      M341  ; 進料夾爪夾持手動
      OR      M241  ; 進料夾爪夾持自動
      OR      Y101  ; 進料夾爪夾持SV
      ANI     M340  ; 進料夾爪開夾手動
      ANI     M240  ; 進料夾爪開夾自動
      OR      M235  ; 主傳動強制夾持
      OR      M238  ; ROBOT異常進料夾爪復歸
      OUT     Y101  ; 進料夾爪夾持SV
88    LD      Y100  ; 進料夾爪開夾SV
      AND     SM412  ; 1S CLOCK
      OR      X2  ; 進料夾爪--開定點
      OUT     M116  ; 進料夾爪開夾PB燈
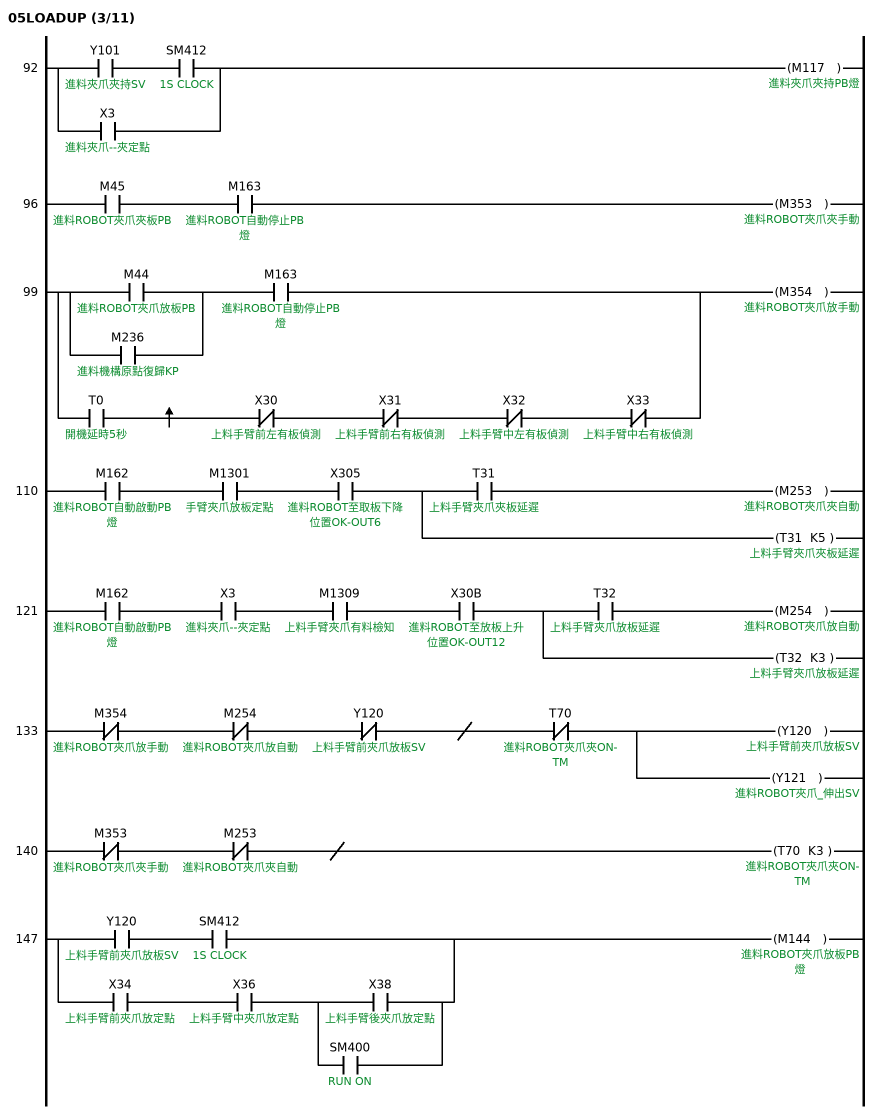
92    LD      Y101  ; 進料夾爪夾持SV
      AND     SM412  ; 1S CLOCK
      OR      X3  ; 進料夾爪--夾定點
      OUT     M117  ; 進料夾爪夾持PB燈
96    LD      M45  ; 進料ROBOT夾爪夾板PB
      AND     M163  ; 進料ROBOT自動停止PB燈
      OUT     M353  ; 進料ROBOT夾爪夾手動
99    LD      M44  ; 進料ROBOT夾爪放板PB
      OR      M236  ; 進料機構原點復歸KP
      AND     M163  ; 進料ROBOT自動停止PB燈
      LD      T0  ; 開機延時5秒
      MEP
      ANI     X30  ; 上料手臂前左有板偵測
      ANI     X31  ; 上料手臂前右有板偵測
      ANI     X32  ; 上料手臂中左有板偵測
      ANI     X33  ; 上料手臂中右有板偵測
      ORB
      OUT     M354  ; 進料ROBOT夾爪放手動
110   LD      M162  ; 進料ROBOT自動啟動PB燈
      AND     M1301  ; 手臂夾爪放板定點
      AND     X305  ; 進料ROBOT至取板下降位置OK-OUT6
      MPS
      AND     T31  ; 上料手臂夾爪夾板延遲
      OUT     M253  ; 進料ROBOT夾爪夾自動
      MPP
      OUT     T31 K5  ; 上料手臂夾爪夾板延遲
121   LD      M162  ; 進料ROBOT自動啟動PB燈
      AND     X3  ; 進料夾爪--夾定點
      AND     M1309  ; 上料手臂夾爪有料檢知
      AND     X30B  ; 進料ROBOT至放板上升位置OK-OUT12
      MPS
      AND     T32  ; 上料手臂夾爪放板延遲
      OUT     M254  ; 進料ROBOT夾爪放自動
      MPP
      OUT     T32 K3  ; 上料手臂夾爪放板延遲
133   LDI     M354  ; 進料ROBOT夾爪放手動
      ANI     M254  ; 進料ROBOT夾爪放自動
      ANI     Y120  ; 上料手臂前夾爪放板SV
      INV
      ANI     T70  ; 進料ROBOT夾爪夾ON-TM
      OUT     Y120  ; 上料手臂前夾爪放板SV
      OUT     Y121  ; 進料ROBOT夾爪_伸出SV
140   LDI     M353  ; 進料ROBOT夾爪夾手動
      ANI     M253  ; 進料ROBOT夾爪夾自動
      INV
      OUT     T70 K3  ; 進料ROBOT夾爪夾ON-TM
147   LD      Y120  ; 上料手臂前夾爪放板SV
      AND     SM412  ; 1S CLOCK
      LD      X34  ; 上料手臂前夾爪放定點
      AND     X36  ; 上料手臂中夾爪放定點
      LD      X38  ; 上料手臂後夾爪放定點
      OR      SM400  ; RUN ON
      ANB
      ORB
      OUT     M144  ; 進料ROBOT夾爪放板PB燈
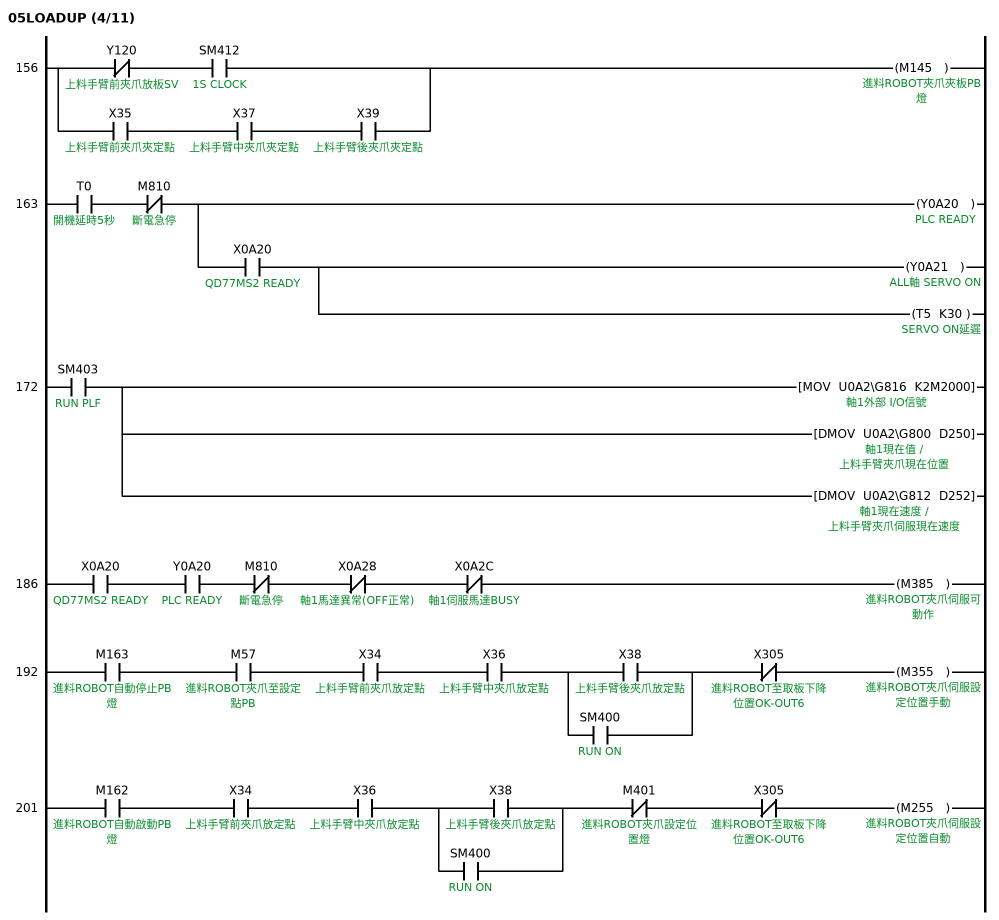
156   LDI     Y120  ; 上料手臂前夾爪放板SV
      AND     SM412  ; 1S CLOCK
      LD      X35  ; 上料手臂前夾爪夾定點
      AND     X37  ; 上料手臂中夾爪夾定點
      AND     X39  ; 上料手臂後夾爪夾定點
      ORB
      OUT     M145  ; 進料ROBOT夾爪夾板PB燈
163   LD      T0  ; 開機延時5秒
      ANI     M810  ; 斷電急停
      OUT     Y0A20  ; PLC READY
      AND     X0A20  ; QD77MS2 READY
      OUT     Y0A21  ; ALL軸 SERVO ON
      OUT     T5 K30  ; SERVO ON延遲
172   LD      SM403  ; RUN PLF
      MOV     U0A2\G816 K2M2000  ; 軸1外部 I/O信號 / 軸1伺服馬達外極限
      DMOV    U0A2\G800 D250  ; 軸1現在值
      DMOV    U0A2\G812 D252  ; 軸1現在速度 / 上料手臂夾爪伺服現在速度
186   LD      X0A20  ; QD77MS2 READY
      AND     Y0A20  ; PLC READY
      ANI     M810  ; 斷電急停
      ANI     X0A28  ; 軸1馬達異常(OFF正常)
      ANI     X0A2C  ; 軸1伺服馬達BUSY
      OUT     M385  ; 進料ROBOT夾爪伺服可動作
192   LD      M163  ; 進料ROBOT自動停止PB燈
      AND     M57  ; 進料ROBOT夾爪至設定點PB
      AND     X34  ; 上料手臂前夾爪放定點
      AND     X36  ; 上料手臂中夾爪放定點
      LD      X38  ; 上料手臂後夾爪放定點
      OR      SM400  ; RUN ON
      ANB
      ANI     X305  ; 進料ROBOT至取板下降位置OK-OUT6
      OUT     M355  ; 進料ROBOT夾爪伺服設定位置手動
201   LD      M162  ; 進料ROBOT自動啟動PB燈
      AND     X34  ; 上料手臂前夾爪放定點
      AND     X36  ; 上料手臂中夾爪放定點
      LD      X38  ; 上料手臂後夾爪放定點
      OR      SM400  ; RUN ON
      ANB
      ANI     M401  ; 進料ROBOT夾爪設定位置燈
      ANI     X305  ; 進料ROBOT至取板下降位置OK-OUT6
      OUT     M255  ; 進料ROBOT夾爪伺服設定位置自動
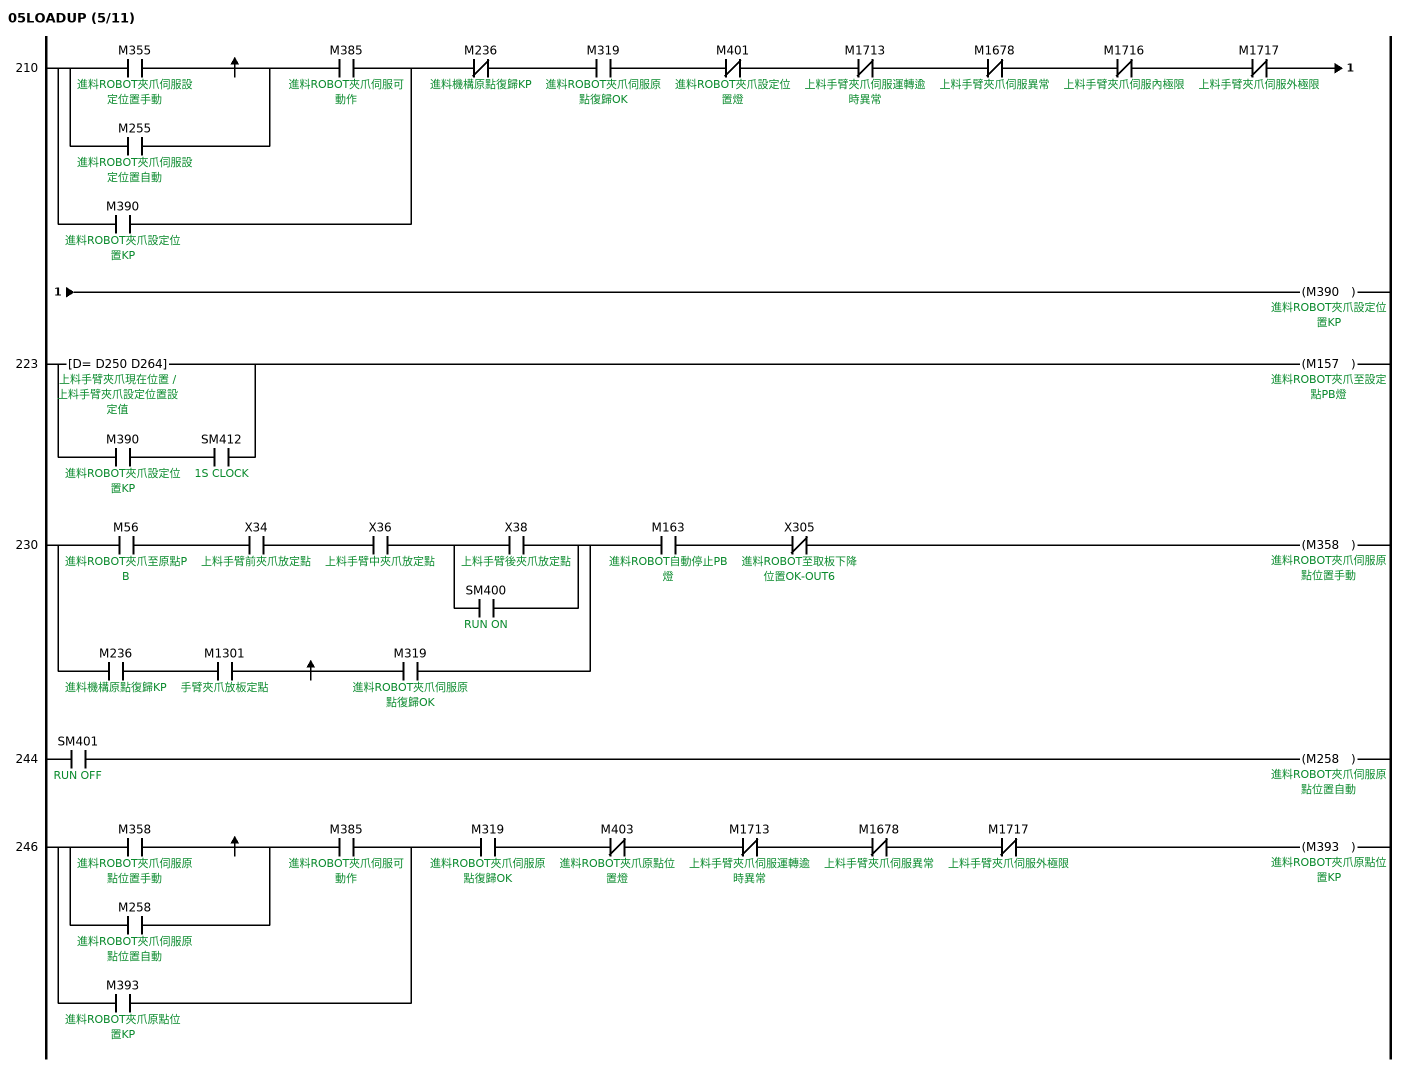
210   LD      M355  ; 進料ROBOT夾爪伺服設定位置手動
      MEP
      OR      M255  ; 進料ROBOT夾爪伺服設定位置自動
      AND     M385  ; 進料ROBOT夾爪伺服可動作
      OR      M390  ; 進料ROBOT夾爪設定位置KP
      ANI     M236  ; 進料機構原點復歸KP
      AND     M319  ; 進料ROBOT夾爪伺服原點復歸OK
      ANI     M401  ; 進料ROBOT夾爪設定位置燈
      ANI     M1713  ; 上料手臂夾爪伺服運轉逾時異常
      ANI     M1678  ; 上料手臂夾爪伺服異常
      ANI     M1716  ; 上料手臂夾爪伺服內極限
      ANI     M1717  ; 上料手臂夾爪伺服外極限
      OUT     M390  ; 進料ROBOT夾爪設定位置KP
223   LDD=    D250 D264  ; 上料手臂夾爪現在位置 / 上料手臂夾爪設定位置設定值
      LD      M390  ; 進料ROBOT夾爪設定位置KP
      AND     SM412  ; 1S CLOCK
      ORB
      OUT     M157  ; 進料ROBOT夾爪至設定點PB燈
230   LD      M56  ; 進料ROBOT夾爪至原點PB
      AND     X34  ; 上料手臂前夾爪放定點
      AND     X36  ; 上料手臂中夾爪放定點
      LD      X38  ; 上料手臂後夾爪放定點
      OR      SM400  ; RUN ON
      ANB
      LD      M236  ; 進料機構原點復歸KP
      AND     M1301  ; 手臂夾爪放板定點
      MEP
      AND     M319  ; 進料ROBOT夾爪伺服原點復歸OK
      ORB
      AND     M163  ; 進料ROBOT自動停止PB燈
      ANI     X305  ; 進料ROBOT至取板下降位置OK-OUT6
      OUT     M358  ; 進料ROBOT夾爪伺服原點位置手動
244   LD      SM401  ; RUN OFF
      OUT     M258  ; 進料ROBOT夾爪伺服原點位置自動
246   LD      M358  ; 進料ROBOT夾爪伺服原點位置手動
      MEP
      OR      M258  ; 進料ROBOT夾爪伺服原點位置自動
      AND     M385  ; 進料ROBOT夾爪伺服可動作
      OR      M393  ; 進料ROBOT夾爪原點位置KP
      AND     M319  ; 進料ROBOT夾爪伺服原點復歸OK
      ANI     M403  ; 進料ROBOT夾爪原點位置燈
      ANI     M1713  ; 上料手臂夾爪伺服運轉逾時異常
      ANI     M1678  ; 上料手臂夾爪伺服異常
      ANI     M1717  ; 上料手臂夾爪伺服外極限
      OUT     M393  ; 進料ROBOT夾爪原點位置KP
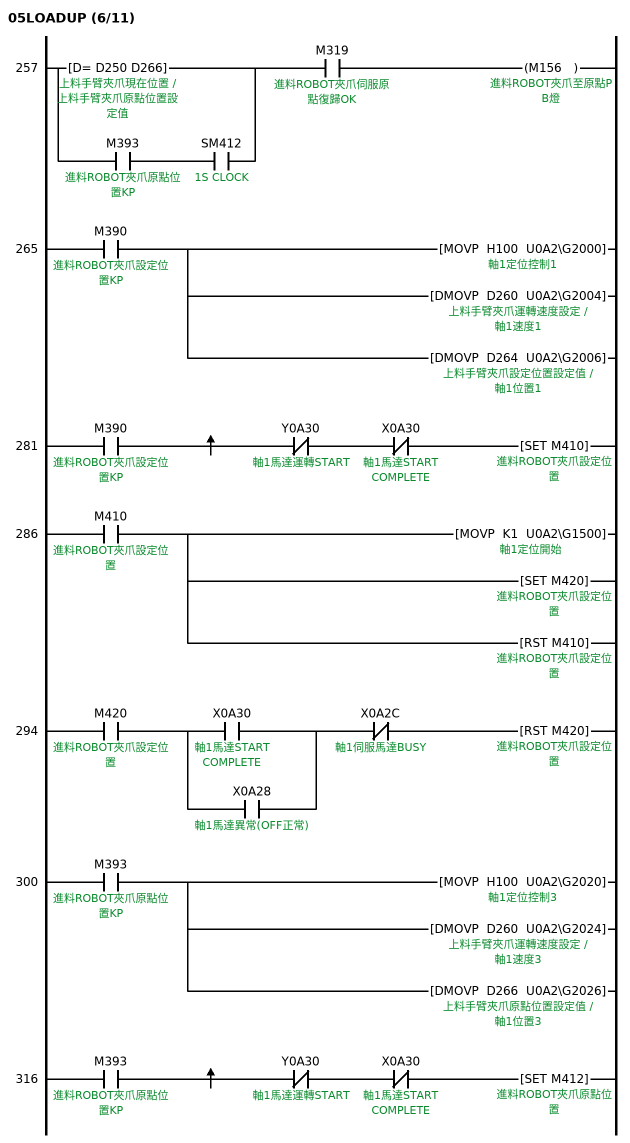
257   LDD=    D250 D266  ; 上料手臂夾爪現在位置 / 上料手臂夾爪原點位置設定值
      LD      M393  ; 進料ROBOT夾爪原點位置KP
      AND     SM412  ; 1S CLOCK
      ORB
      AND     M319  ; 進料ROBOT夾爪伺服原點復歸OK
      OUT     M156  ; 進料ROBOT夾爪至原點PB燈
265   LD      M390  ; 進料ROBOT夾爪設定位置KP
      MOVP    H100 U0A2\G2000  ; 軸1定位控制1
      DMOVP   D260 U0A2\G2004  ; 上料手臂夾爪運轉速度設定 / 軸1速度1
      DMOVP   D264 U0A2\G2006  ; 軸1位置1
281   LD      M390  ; 進料ROBOT夾爪設定位置KP
      MEP
      ANI     Y0A30  ; 軸1馬達運轉START
      ANI     X0A30  ; 軸1馬達START COMPLETE
      SET     M410  ; 進料ROBOT夾爪設定位置
286   LD      M410  ; 進料ROBOT夾爪設定位置
      MOVP    K1 U0A2\G1500  ; 軸1定位開始
      SET     M420  ; 進料ROBOT夾爪設定位置
      RST     M410  ; 進料ROBOT夾爪設定位置
294   LD      M420  ; 進料ROBOT夾爪設定位置
      LD      X0A30  ; 軸1馬達START COMPLETE
      OR      X0A28  ; 軸1馬達異常(OFF正常)
      ANB
      ANI     X0A2C  ; 軸1伺服馬達BUSY
      RST     M420  ; 進料ROBOT夾爪設定位置
300   LD      M393  ; 進料ROBOT夾爪原點位置KP
      MOVP    H100 U0A2\G2020  ; 軸1定位控制3
      DMOVP   D260 U0A2\G2024  ; 軸1速度3
      DMOVP   D266 U0A2\G2026  ; 軸1位置3
316   LD      M393  ; 進料ROBOT夾爪原點位置KP
      MEP
      ANI     Y0A30  ; 軸1馬達運轉START
      ANI     X0A30  ; 軸1馬達START COMPLETE
      SET     M412  ; 進料ROBOT夾爪原點位置
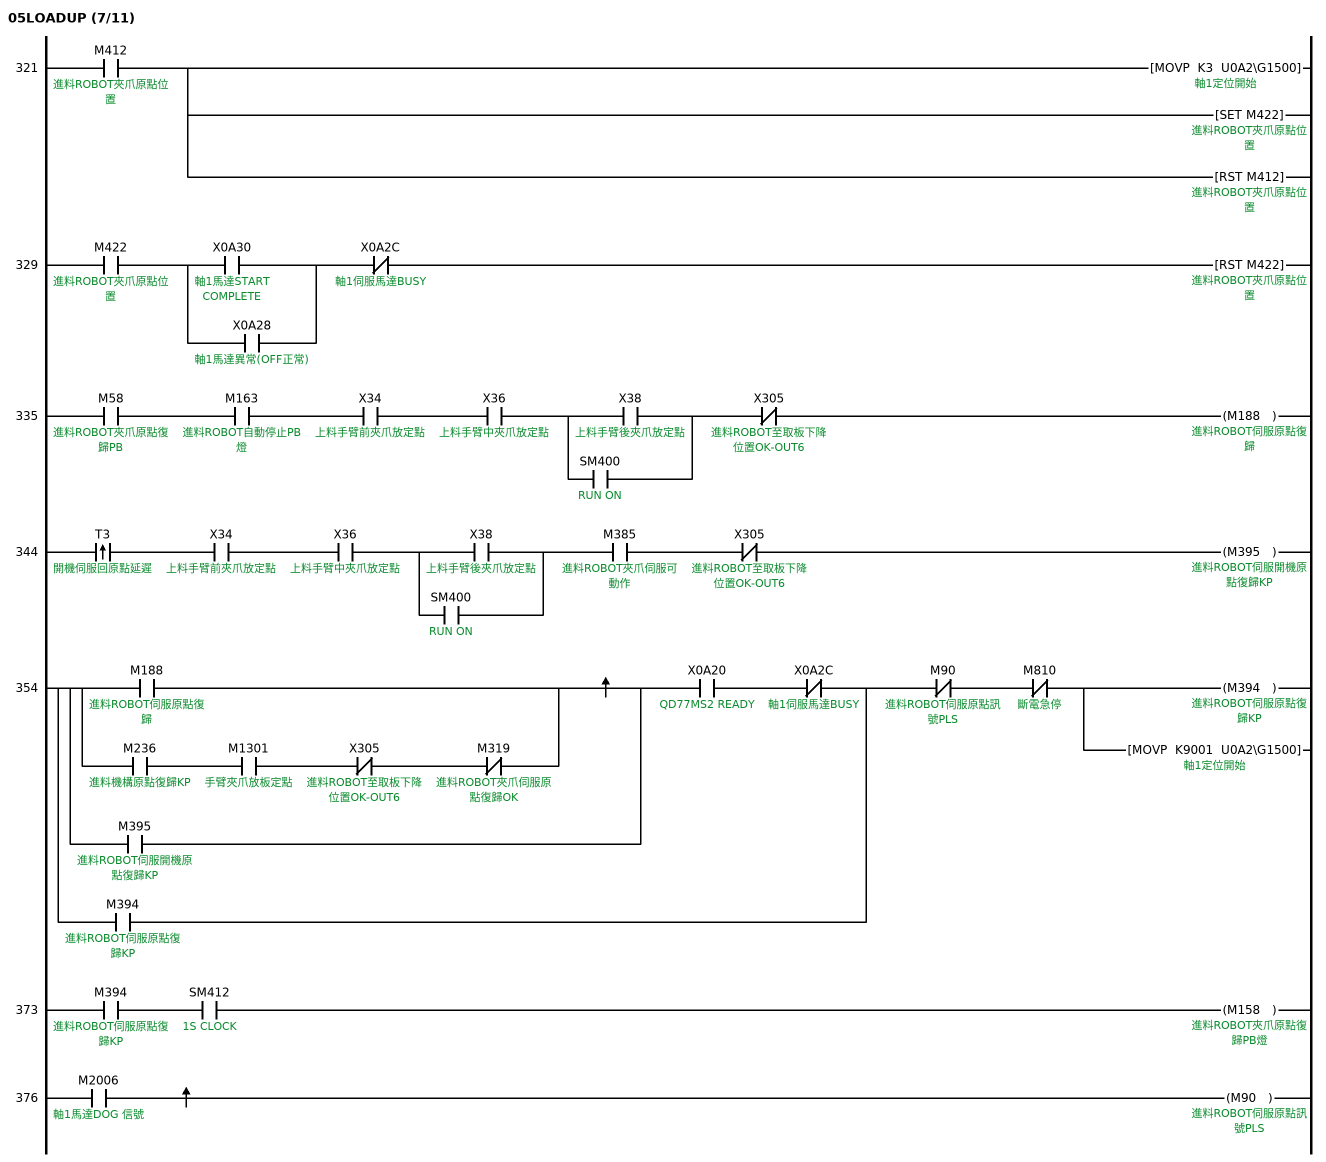
321   LD      M412  ; 進料ROBOT夾爪原點位置
      MOVP    K3 U0A2\G1500
      SET     M422  ; 進料ROBOT夾爪原點位置
      RST     M412  ; 進料ROBOT夾爪原點位置
329   LD      M422  ; 進料ROBOT夾爪原點位置
      LD      X0A30  ; 軸1馬達START COMPLETE
      OR      X0A28  ; 軸1馬達異常(OFF正常)
      ANB
      ANI     X0A2C  ; 軸1伺服馬達BUSY
      RST     M422  ; 進料ROBOT夾爪原點位置
335   LD      M58  ; 進料ROBOT夾爪原點復歸PB
      AND     M163  ; 進料ROBOT自動停止PB燈
      AND     X34  ; 上料手臂前夾爪放定點
      AND     X36  ; 上料手臂中夾爪放定點
      LD      X38  ; 上料手臂後夾爪放定點
      OR      SM400  ; RUN ON
      ANB
      ANI     X305  ; 進料ROBOT至取板下降位置OK-OUT6
      OUT     M188  ; 進料ROBOT伺服原點復歸
344   LDP     T3  ; 開機伺服回原點延遲
      AND     X34  ; 上料手臂前夾爪放定點
      AND     X36  ; 上料手臂中夾爪放定點
      LD      X38  ; 上料手臂後夾爪放定點
      OR      SM400  ; RUN ON
      ANB
      AND     M385  ; 進料ROBOT夾爪伺服可動作
      ANI     X305  ; 進料ROBOT至取板下降位置OK-OUT6
      OUT     M395  ; 進料ROBOT伺服開機原點復歸KP
354   LD      M188  ; 進料ROBOT伺服原點復歸
      LD      M236  ; 進料機構原點復歸KP
      AND     M1301  ; 手臂夾爪放板定點
      ANI     X305  ; 進料ROBOT至取板下降位置OK-OUT6
      ANI     M319  ; 進料ROBOT夾爪伺服原點復歸OK
      ORB
      MEP
      OR      M395  ; 進料ROBOT伺服開機原點復歸KP
      AND     X0A20  ; QD77MS2 READY
      ANI     X0A2C  ; 軸1伺服馬達BUSY
      OR      M394  ; 進料ROBOT伺服原點復歸KP
      ANI     M90  ; 進料ROBOT伺服原點訊號PLS
      ANI     M810  ; 斷電急停
      OUT     M394  ; 進料ROBOT伺服原點復歸KP
      MOVP    K9001 U0A2\G1500
373   LD      M394  ; 進料ROBOT伺服原點復歸KP
      AND     SM412  ; 1S CLOCK
      OUT     M158  ; 進料ROBOT夾爪原點復歸PB燈
376   LD      M2006  ; 軸1馬達DOG 信號
      MEP
      OUT     M90  ; 進料ROBOT伺服原點訊號PLS
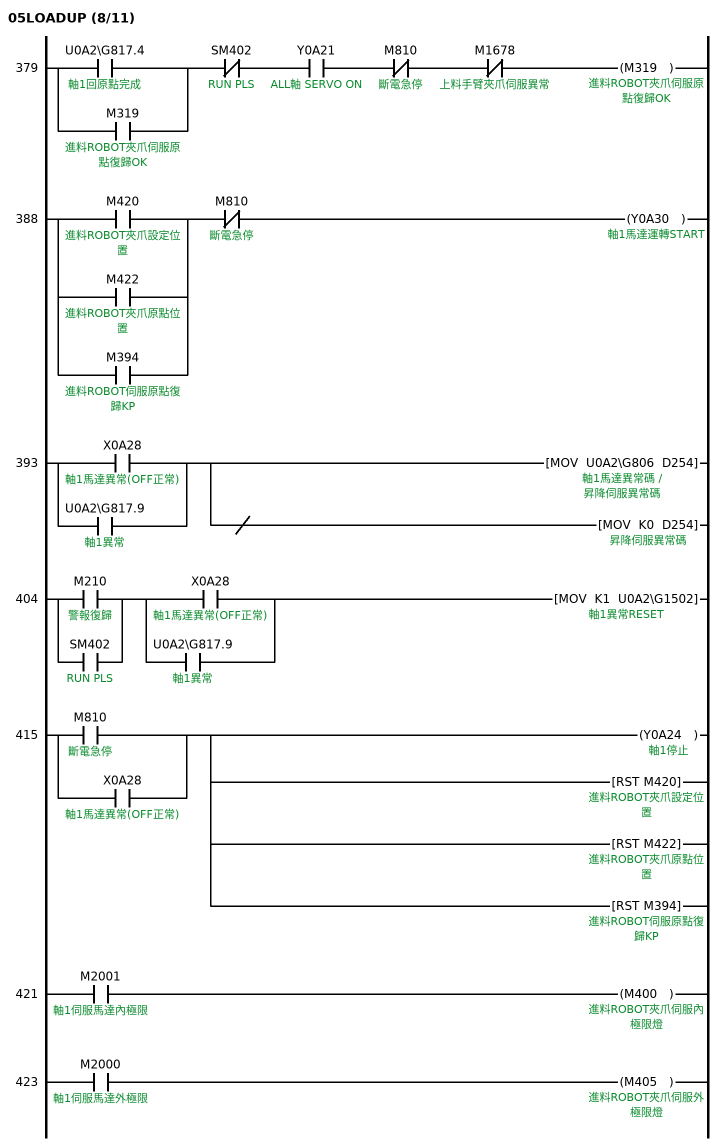
379   LD      U0A2\G817.4  ; 軸1回原點完成
      OR      M319  ; 進料ROBOT夾爪伺服原點復歸OK
      ANI     SM402  ; RUN PLS
      AND     Y0A21  ; ALL軸 SERVO ON
      ANI     M810  ; 斷電急停
      ANI     M1678  ; 上料手臂夾爪伺服異常
      OUT     M319  ; 進料ROBOT夾爪伺服原點復歸OK
388   LD      M420  ; 進料ROBOT夾爪設定位置
      OR      M422  ; 進料ROBOT夾爪原點位置
      OR      M394  ; 進料ROBOT伺服原點復歸KP
      ANI     M810  ; 斷電急停
      OUT     Y0A30  ; 軸1馬達運轉START
393   LD      X0A28  ; 軸1馬達異常(OFF正常)
      OR      U0A2\G817.9  ; 軸1異常
      MOV     U0A2\G806 D254  ; 軸1馬達異常碼 / 昇降伺服異常碼
      INV
      MOV     K0 D254
404   LD      M210  ; 警報復歸
      OR      SM402  ; RUN PLS
      LD      X0A28  ; 軸1馬達異常(OFF正常)
      OR      U0A2\G817.9  ; 軸1異常
      ANB
      MOV     K1 U0A2\G1502  ; 軸1異常RESET
415   LD      M810  ; 斷電急停
      OR      X0A28  ; 軸1馬達異常(OFF正常)
      OUT     Y0A24  ; 軸1停止
      RST     M420  ; 進料ROBOT夾爪設定位置
      RST     M422  ; 進料ROBOT夾爪原點位置
      RST     M394  ; 進料ROBOT伺服原點復歸KP
421   LD      M2001  ; 軸1伺服馬達內極限
      OUT     M400  ; 進料ROBOT夾爪伺服內極限燈
423   LD      M2000  ; 軸1伺服馬達外極限
      OUT     M405  ; 進料ROBOT夾爪伺服外極限燈
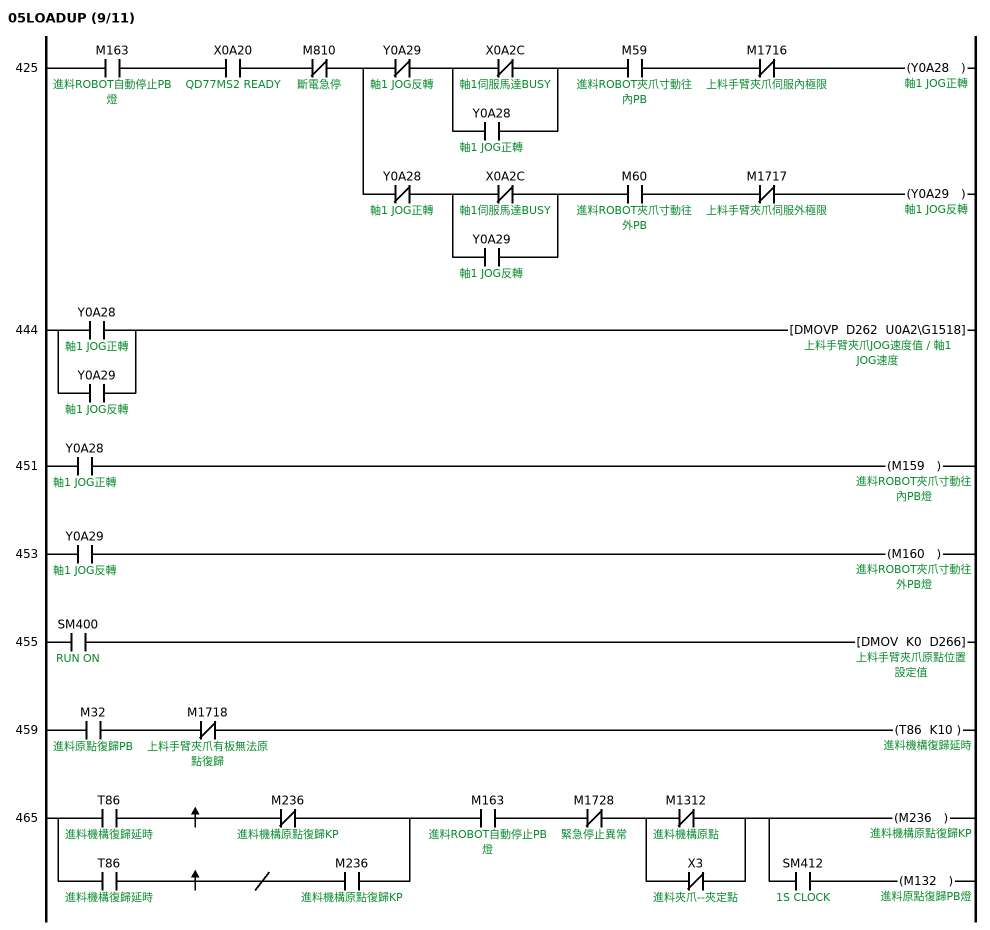
425   LD      M163  ; 進料ROBOT自動停止PB燈
      AND     X0A20  ; QD77MS2 READY
      ANI     M810  ; 斷電急停
      MPS
      ANI     Y0A29  ; 軸1 JOG反轉
      LDI     X0A2C  ; 軸1伺服馬達BUSY
      OR      Y0A28  ; 軸1 JOG正轉
      ANB
      AND     M59  ; 進料ROBOT夾爪寸動往內PB
      ANI     M1716  ; 上料手臂夾爪伺服內極限
      OUT     Y0A28  ; 軸1 JOG正轉
      MPP
      ANI     Y0A28  ; 軸1 JOG正轉
      LDI     X0A2C  ; 軸1伺服馬達BUSY
      OR      Y0A29  ; 軸1 JOG反轉
      ANB
      AND     M60  ; 進料ROBOT夾爪寸動往外PB
      ANI     M1717  ; 上料手臂夾爪伺服外極限
      OUT     Y0A29  ; 軸1 JOG反轉
444   LD      Y0A28  ; 軸1 JOG正轉
      OR      Y0A29  ; 軸1 JOG反轉
      DMOVP   D262 U0A2\G1518  ; 上料手臂夾爪JOG速度值 / 軸1 JOG速度
451   LD      Y0A28  ; 軸1 JOG正轉
      OUT     M159  ; 進料ROBOT夾爪寸動往內PB燈
453   LD      Y0A29  ; 軸1 JOG反轉
      OUT     M160  ; 進料ROBOT夾爪寸動往外PB燈
455   LD      SM400  ; RUN ON
      DMOV    K0 D266
459   LD      M32  ; 進料原點復歸PB
      ANI     M1718  ; 上料手臂夾爪有板無法原點復歸
      OUT     T86 K10  ; 進料機構復歸延時
465   LD      T86  ; 進料機構復歸延時
      MEP
      ANI     M236  ; 進料機構原點復歸KP
      LD      T86  ; 進料機構復歸延時
      MEP
      INV
      AND     M236  ; 進料機構原點復歸KP
      ORB
      AND     M163  ; 進料ROBOT自動停止PB燈
      ANI     M1728  ; 緊急停止異常
      LDI     M1312  ; 進料機構原點
      ORI     X3  ; 進料夾爪--夾定點
      ANB
      OUT     M236  ; 進料機構原點復歸KP
      AND     SM412  ; 1S CLOCK
      OUT     M132  ; 進料原點復歸PB燈
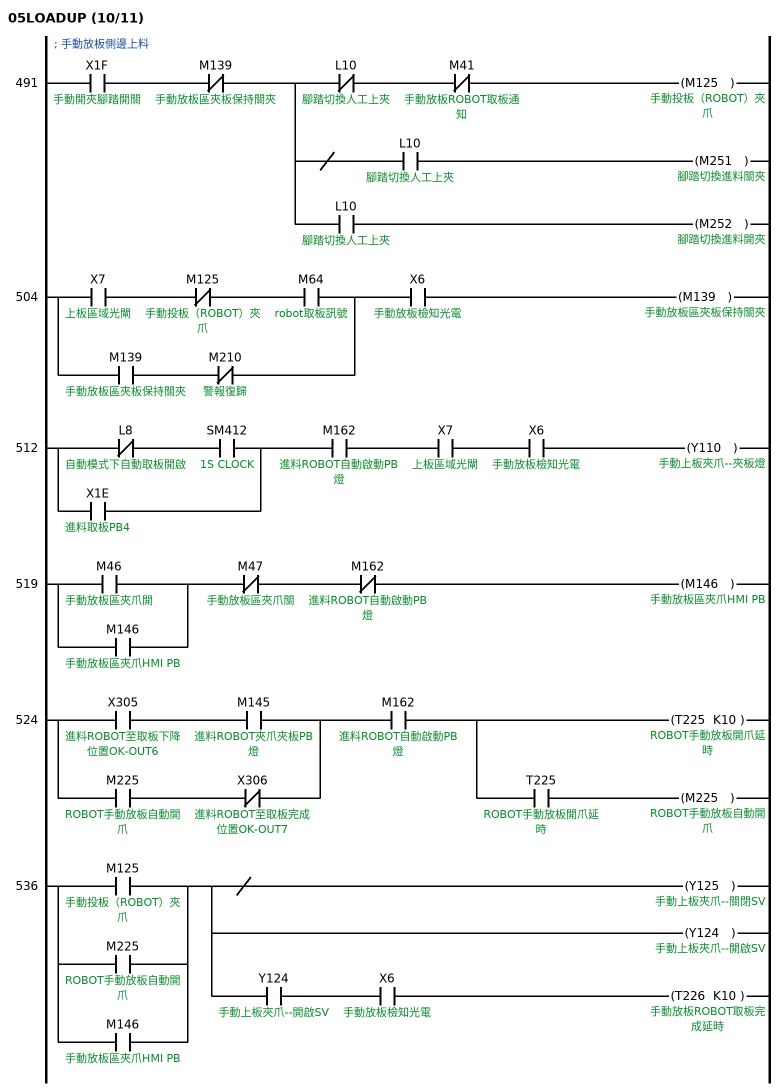
; 手動放板側邊上料
491   LD      X1F  ; 手動開夾腳踏開關
      ANI     M139  ; 手動放板區夾板保持關夾
      MPS
      ANI     L10  ; 腳踏切換人工上夾
      ANI     M41  ; 手動放板ROBOT取板通知
      OUT     M125  ; 手動投板（ROBOT）夾爪
      MRD
      INV
      AND     L10  ; 腳踏切換人工上夾
      OUT     M251  ; 腳踏切換進料關夾
      MPP
      AND     L10  ; 腳踏切換人工上夾
      OUT     M252  ; 腳踏切換進料開夾
504   LD      X7  ; 上板區域光閘
      ANI     M125  ; 手動投板（ROBOT）夾爪
      AND     M64  ; robot取板訊號
      LD      M139  ; 手動放板區夾板保持關夾
      ANI     M210  ; 警報復歸
      ORB
      AND     X6  ; 手動放板檢知光電
      OUT     M139  ; 手動放板區夾板保持關夾
512   LDI     L8  ; 自動模式下自動取板開啟
      AND     SM412  ; 1S CLOCK
      OR      X1E  ; 進料取板PB4
      AND     M162  ; 進料ROBOT自動啟動PB燈
      AND     X7  ; 上板區域光閘
      AND     X6  ; 手動放板檢知光電
      OUT     Y110  ; 手動上板夾爪--夾板燈
519   LD      M46  ; 手動放板區夾爪開
      OR      M146  ; 手動放板區夾爪HMI PB
      ANI     M47  ; 手動放板區夾爪關
      ANI     M162  ; 進料ROBOT自動啟動PB燈
      OUT     M146  ; 手動放板區夾爪HMI PB
524   LD      X305  ; 進料ROBOT至取板下降位置OK-OUT6
      AND     M145  ; 進料ROBOT夾爪夾板PB燈
      LD      M225  ; ROBOT手動放板自動開爪
      ANI     X306  ; 進料ROBOT至取板完成位置OK-OUT7
      ORB
      AND     M162  ; 進料ROBOT自動啟動PB燈
      OUT     T225 K10  ; ROBOT手動放板開爪延時
      AND     T225  ; ROBOT手動放板開爪延時
      OUT     M225  ; ROBOT手動放板自動開爪
536   LD      M125  ; 手動投板（ROBOT）夾爪
      OR      M225  ; ROBOT手動放板自動開爪
      OR      M146  ; 手動放板區夾爪HMI PB
      MPS
      INV
      OUT     Y125  ; 手動上板夾爪--關閉SV
      MPP
      OUT     Y124  ; 手動上板夾爪--開啟SV
      AND     Y124  ; 手動上板夾爪--開啟SV
      AND     X6  ; 手動放板檢知光電
      OUT     T226 K10  ; 手動放板ROBOT取板完成延時
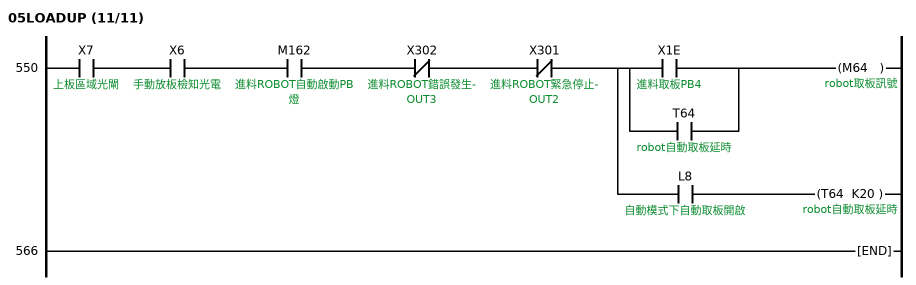
550   LD      X7  ; 上板區域光閘
      AND     X6  ; 手動放板檢知光電
      AND     M162  ; 進料ROBOT自動啟動PB燈
      ANI     X302  ; 進料ROBOT錯誤發生-OUT3
      ANI     X301  ; 進料ROBOT緊急停止-OUT2
      MPS
      LD      X1E  ; 進料取板PB4
      OR      T64  ; robot自動取板延時
      ANB
      OUT     M64  ; robot取板訊號
      MPP
      AND     L8  ; 自動模式下自動取板開啟
      OUT     T64 K20  ; robot自動取板延時
566   END
END_PROGRAM

PROGRAM 06UNLOAD
